# B&R Automation Studio project TD52 (part 71)

#### lIP_EGTCtr.typ
```iecst
TYPE

   tEGTCtr_In : STRUCT
        rT_EG_MaxLim : REAL; (*Exhaust temperature shut down limit from Diane Parameter [°C]*)
        rT_EG_Max : REAL; (*Maximum actual exhaust temperature among all cylinders [°C]*)
        bReset : BOOL; (*Reset of exhaust temperature controller integrator [boolean]*)
        rCA_Init : REAL; (*Reset value of exhaust temperature controller integrator [°CA]*)
        rCA_IP_Act_Rel : REAL; (*External actual ignition timing offset [°CA]*)
    END_STRUCT;

   tEGTCtr_Out : STRUCT
        ulim : REAL; (*Limited controller output [°CA] oldname: ITOffuLim*)
        u : REAL; (*Unlimited controller output [°CA] oldname: ITOffu*)
        up : REAL; (*Unlimited proportional controller output [°CA] oldname: ITOffup*)
        ui : REAL; (*Unlimited integral controller output [°CA] oldname: ITOffui*)
        ud : REAL; (*Unlimited derivative controller output [°CA] oldname: ITOffud*)
        e : REAL; (*Control error without anti-windup [°C] oldname: ITOffe*)
        AW : REAL; (*Anti-windup feedback error [°C] oldname: ITOffAW*)
    END_STRUCT;

   tEGTCtr_Perm : STRUCT
        rT_EG_DltLim : REAL; (*Delta margin from exhaust temperature limit [°C] oldname: TExhLimCntMar*)
        Kp : REAL; (*Proportional gain of exhaust limit controller [°CA/°C]*)
        Ki : REAL; (*Integral gain of exhaust limit controller [°CA/°C/s]*)
        Kd : REAL; (*Derivative gain of exhaust limit controller [°CA*s/°C]*)
        N : REAL; (*Filter constant for derivative controller gain [1/s]*)
        UpLim : REAL; (*Upper limit for controller output [CAD]*)
        LoLim : REAL; (*Lower limit for controller output [°CA]*)
        KAW : REAL; (*Anti windup gain for exhaust temperature controller integrator [°C/°CA]*)
        DeadLoD : REAL; (*Lower deadband limit for derivative part [°C]*)
        DeadUpD : REAL; (*Upper deadband limit for derivative part [°C]*)
    END_STRUCT;
END_TYPE
TYPE
BlockIO_IP_EGTCtr : STRUCT
	perm : tEGTCtr_Perm;
	BusCreator : tEGTCtr_Out;
	in : tEGTCtr_In;
END_STRUCT;
D_Work_IP_EGTCtr : STRUCT
	DiscreteTimeIntegrator_DSTATE : REAL;
	DiscreteTimeIntegrator1_DSTATE : REAL;
	DiscreteTimeIntegrator_PrevRese : SINT;
	DiscreteTimeIntegrator1_PrevRes : SINT;
	DiscreteTimeIntegrator_IC_LOADI : USINT;
END_STRUCT;
END_TYPE
```

#### IP_EGTCtr.h
```c
/********************************************************************
 * COPYRIGHT -- Bernecker + Rainer Industrie-Elektronik Ges.m.b.H.
 ********************************************************************
 * Program: IP_EGTCtr
 * File: IP_EGTCtr.h
 * Author: 302013638
 * Created: Fri Sep 10 20:20:48 2010
 ********************************************************************
 * Header for program IP_EGTCtr
 ********************************************************************
 * Generated with B&R Automation Studio Target for Simulink V4.2
 * (ERT based)
 ********************************************************************/

#ifndef RTW_HEADER_IP_EGTCtr_h_
#define RTW_HEADER_IP_EGTCtr_h_
#ifndef IP_EGTCtr_COMMON_INCLUDES_
# define IP_EGTCtr_COMMON_INCLUDES_
#include "rtwtypes.h"
#endif                                 /* IP_EGTCtr_COMMON_INCLUDES_ */

#include "IP_EGTCtr_types.h"
#include "lIP_EGTCtr.h"

/* Macros for accessing real-time model data structure */
#ifndef rtmGetErrorStatus
# define rtmGetErrorStatus(rtm)        ((void*) 0)
#endif

#ifndef rtmSetErrorStatus
# define rtmSetErrorStatus(rtm, val)   ((void) 0)
#endif

#ifndef rtmGetStopRequested
# define rtmGetStopRequested(rtm)      ((void*) 0)
#endif

#ifndef MIN
#define MIN(a,b)                       ((a) < (b) ? (a) : (b))
#endif

#ifndef MAX
#define MAX(a,b)                       ((a) > (b) ? (a) : (b))
#endif

/* Block signals (auto storage) */

/* Block states (auto storage) for system '<Root>' */

/* Block signals (auto storage) */
extern BlockIO_IP_EGTCtr IP_EGTCtr_B;

/* Block states (auto storage) */
extern D_Work_IP_EGTCtr IP_EGTCtr_DWork;

/* Model entry point functions */
extern void IP_EGTCtr_initialize(struct fIP_EGTCtr* inst);
extern void IP_EGTCtr_step(struct fIP_EGTCtr* inst);
extern void IP_EGTCtr_terminate(struct fIP_EGTCtr* inst);

/*-
 * The generated code includes comments that allow you to trace directly
 * back to the appropriate location in the model.  The basic format
 * is <system>/block_name, where system is the system number (uniquely
 * assigned by Simulink) and block_name is the name of the block.
 *
 * Use the MATLAB hilite_system command to trace the generated code back
 * to the model.  For example,
 *
 * hilite_system('<S3>')    - opens system 3
 * hilite_system('<S3>/Kp') - opens and selects block Kp which resides in S3
 *
 * Here is the system hierarchy for this model
 *
 * '<Root>' : 'IP_EGTCtr'
 * '<S1>'   : 'IP_EGTCtr/DocBlock'
 * '<S2>'   : 'IP_EGTCtr/Model Info'
 * '<S3>'   : 'IP_EGTCtr/TexhCntrSys'
 * '<S4>'   : 'IP_EGTCtr/TexhCntrSys/Dead Zone Dynamic'
 * '<S5>'   : 'IP_EGTCtr/TexhCntrSys/Saturation Dynamic4'
 */
#endif                                 /* RTW_HEADER_IP_EGTCtr_h_ */
```

#### IP_EGTCtr_private.h
```c
/********************************************************************
 * COPYRIGHT -- Bernecker + Rainer Industrie-Elektronik Ges.m.b.H.
 ********************************************************************
 * Program: IP_EGTCtr
 * File: IP_EGTCtr_private.h
 * Author: 302013638
 * Created: Fri Sep 10 20:20:48 2010
 ********************************************************************
 * Header for program IP_EGTCtr
 ********************************************************************
 * Generated with B&R Automation Studio Target for Simulink V4.2
 * (ERT based)
 ********************************************************************/

#ifndef RTW_HEADER_IP_EGTCtr_private_h_
#define RTW_HEADER_IP_EGTCtr_private_h_
#include "rtwtypes.h"
#include <bur/plctypes.h>
#ifndef __RTWTYPES_H__
#error This file requires rtwtypes.h to be included
#else
#ifdef TMWTYPES_PREVIOUSLY_INCLUDED
#error This file requires rtwtypes.h to be included before tmwtypes.h
#else

/* Check for inclusion of an incorrect version of rtwtypes.h */
#ifndef RTWTYPES_ID_C08S16I32L32N32F1
#error This code was generated with a different "rtwtypes.h" than the file included
#endif                                 /* RTWTYPES_ID_C08S16I32L32N32F1 */
#endif                                 /* TMWTYPES_PREVIOUSLY_INCLUDED */
#endif                                 /* __RTWTYPES_H__ */

#ifndef MIN
#define MIN(a,b)                       ((a) < (b) ? (a) : (b))
#endif

#ifndef MAX
#define MAX(a,b)                       ((a) > (b) ? (a) : (b))
#endif
#endif                                 /* RTW_HEADER_IP_EGTCtr_private_h_ */
```

#### IP_EGTCtr_types.h
```c
/********************************************************************
 * COPYRIGHT -- Bernecker + Rainer Industrie-Elektronik Ges.m.b.H.
 ********************************************************************
 * Program: IP_EGTCtr
 * File: IP_EGTCtr_types.h
 * Author: 302013638
 * Created: Fri Sep 10 20:20:48 2010
 ********************************************************************
 * Header for program IP_EGTCtr
 ********************************************************************
 * Generated with B&R Automation Studio Target for Simulink V4.2
 * (ERT based)
 ********************************************************************/

#ifndef RTW_HEADER_IP_EGTCtr_types_h_
#define RTW_HEADER_IP_EGTCtr_types_h_
#include "rtwtypes.h"
#ifndef MIN
#define MIN(a,b)                       ((a) < (b) ? (a) : (b))
#endif

#ifndef MAX
#define MAX(a,b)                       ((a) > (b) ? (a) : (b))
#endif

#endif                                 /* RTW_HEADER_IP_EGTCtr_types_h_ */
```

#### rtwtypes.h
```c
/********************************************************************
 * COPYRIGHT -- Bernecker + Rainer Industrie-Elektronik Ges.m.b.H.
 ********************************************************************
 * Program: IP_EGTCtr
 * File: rtwtypes.h
 * Author: 302013638
 * Created: Fri Sep 10 20:20:48 2010
 ********************************************************************
 * Header for program IP_EGTCtr
 ********************************************************************
 * Generated with B&R Automation Studio Target for Simulink V4.2
 * (ERT based)
 ********************************************************************/

#ifndef __RTWTYPES_H__
#define __RTWTYPES_H__
#ifndef TRUE
# define TRUE                          (1U)
#endif

#ifndef FALSE
# define FALSE                         (0U)
#endif

#ifndef __TMWTYPES__
#define __TMWTYPES__
#include <limits.h>

/*=======================================================================*
 * Target hardware information
 *   Device type: Intel->x86/Pentium
 *   Number of bits:     char:   8    short:   16    long:  32
 *                       long:  32
 *                       native word size:  32
 *   Byte ordering: LittleEndian
 *   Signed integer division rounds to: Zero
 *   Shift right on a signed integer as arithmetic shift: on
 *=======================================================================*/

/*=======================================================================*
 * Fixed width word size data types:                                     *
 *   int8_T, int16_T, int32_T     - signed 8, 16, or 32 bit integers     *
 *   uint8_T, uint16_T, uint32_T  - unsigned 8, 16, or 32 bit integers   *
 *   real32_T, real64_T           - 32 and 64 bit floating point numbers *
 *=======================================================================*/
typedef signed char int8_T;
typedef unsigned char uint8_T;
typedef short int16_T;
typedef unsigned short uint16_T;
typedef long int32_T;
typedef unsigned long uint32_T;
typedef float real32_T;
typedef double real64_T;

/*===========================================================================*
 * Generic type definitions: real_T, time_T, boolean_T, int_T, uint_T,       *
 *                           ulong_T, char_T and byte_T.                     *
 *===========================================================================*/
typedef double real_T;
typedef double time_T;
typedef unsigned char boolean_T;
typedef long int_T;
typedef unsigned long uint_T;
typedef unsigned long ulong_T;
typedef char char_T;
typedef unsigned char uchar_T;
typedef char_T byte_T;

/*=======================================================================*
 * Min and Max:                                                          *
 *   int8_T, int16_T, int32_T     - signed 8, 16, or 32 bit integers     *
 *   uint8_T, uint16_T, uint32_T  - unsigned 8, 16, or 32 bit integers   *
 *=======================================================================*/
#define MAX_int8_T                     ((int8_T)(127))
#define MIN_int8_T                     ((int8_T)(-128))
#define MAX_uint8_T                    ((uint8_T)(255U))
#define MIN_uint8_T                    ((uint8_T)(0U))
#define MAX_int16_T                    ((int16_T)(32767))
#define MIN_int16_T                    ((int16_T)(-32768))
#define MAX_uint16_T                   ((uint16_T)(65535U))
#define MIN_uint16_T                   ((uint16_T)(0U))
#define MAX_int32_T                    ((int32_T)(2147483647))
#define MIN_int32_T                    ((int32_T)(-2147483647-1))
#define MAX_uint32_T                   ((uint32_T)(0xFFFFFFFFU))
#define MIN_uint32_T                   ((uint32_T)(0U))

/* Logical type definitions */
#if (!defined(__cplusplus)) && (!defined(__true_false_are_keywords))
#  ifndef false
#   define false                       (0U)
#  endif

#  ifndef true
#   define true                        (1U)
#  endif
#endif

/*
 * Simulink Coder assumes the code is compiled on a target using a 2's complement representation
 * for signed integer values.
 */
#if ((SCHAR_MIN + 1) != -SCHAR_MAX)
#error "This code must be compiled using a 2's complement representation for signed integer values"
#endif

/* This ID is used to detect inclusion of an incompatible rtwtypes.h */
#define RTWTYPES_ID_C08S16I32L32N32F1
#else                                  /* __TMWTYPES__ */
#define TMWTYPES_PREVIOUSLY_INCLUDED
#endif                                 /* __TMWTYPES__ */

/* Block D-Work pointer type */
typedef void * pointer_T;

/* Simulink specific types */
#ifndef __SIMSTRUC_TYPES_H__
#define __SIMSTRUC_TYPES_H__

/* Trigger directions: falling, either, and rising */
typedef enum {
  FALLING_ZERO_CROSSING = -1,
  ANY_ZERO_CROSSING = 0,
  RISING_ZERO_CROSSING = 1
} ZCDirection;

/* Previous state of a trigger signal */
typedef uint8_T ZCSigState;

/* Initial value of a trigger zero crossing signal */
#define UNINITIALIZED_ZCSIG            0x03U
#define NEG_ZCSIG                      0x02U
#define POS_ZCSIG                      0x01U
#define ZERO_ZCSIG                     0x00U

/* Current state of a trigger signal */
typedef enum {
  FALLING_ZCEVENT = -1,
  NO_ZCEVENT = 0,
  RISING_ZCEVENT = 1
} ZCEventType;

#endif                                 /* __SIMSTRUC_TYPES_H__ */
#endif                                 /* __RTWTYPES_H__ */

#ifndef MIN
#define MIN(a,b)                       ((a) < (b) ? (a) : (b))
#endif

#ifndef MAX
#define MAX(a,b)                       ((a) > (b) ? (a) : (b))
#endif
```

#### IP_EGTCtr.c
```c
/********************************************************************
 * COPYRIGHT -- Bernecker + Rainer Industrie-Elektronik Ges.m.b.H.
 ********************************************************************
 * Program: IP_EGTCtr
 * File: IP_EGTCtr.c
 * Author: 302013638
 * Created: Fri Sep 10 20:20:48 2010
 ********************************************************************
 * Implementation of program IP_EGTCtr
 ********************************************************************
 * Generated with B&R Automation Studio Target for Simulink V4.2
 * (ERT based)
 ********************************************************************/
#include "IP_EGTCtr.h"
#include "IP_EGTCtr_private.h"

/*  Defines */

/*  Data Types */

/**************************** GLOBAL DATA *************************************/
/*  Definitions */

/* Block signals (auto storage) */
struct BlockIO_IP_EGTCtr IP_EGTCtr_B;

/* Block states (auto storage) */
struct D_Work_IP_EGTCtr IP_EGTCtr_DWork;

/*  Declarations  */

/***************************** FILE SCOPE DATA ********************************/

/*************************** FUNCTIONS ****************************************/

/* Model step function */
void IP_EGTCtr_step(struct fIP_EGTCtr* inst)
{
  /* local block i/o variables */
  boolean_T rtb_bReset;
  real32_T rtb_e;
  real32_T rtb_up;
  real32_T rtb_ud;
  real32_T rtb_Product2;
  real32_T rtb_Add;

  /* S-Function (bur_bus_in): '<Root>/Bus Input2' */
  IP_EGTCtr_B.in = inst->in;

  /* BusSelector: '<Root>/BusConversion_InsertedFor_Bus Creator1_at_inport_1' */
  rtb_bReset = IP_EGTCtr_B.in.bReset;

  /* S-Function (bur_bus_in): '<Root>/Bus Input1' */
  IP_EGTCtr_B.perm = inst->perm;

  /* Gain: '<S3>/Gain' incorporates:
   *  Sum: '<S3>/Add4'
   *  Sum: '<S3>/Add6'
   */
  rtb_e = -((IP_EGTCtr_B.in.rT_EG_MaxLim - IP_EGTCtr_B.perm.rT_EG_DltLim) -
            IP_EGTCtr_B.in.rT_EG_Max);

  /* Product: '<S3>/Product1' */
  rtb_up = rtb_e * IP_EGTCtr_B.perm.Kp;

  /* DiscreteIntegrator: '<S3>/Discrete-Time Integrator' */
  if (IP_EGTCtr_DWork.DiscreteTimeIntegrator_IC_LOADI != 0) {
    IP_EGTCtr_DWork.DiscreteTimeIntegrator_DSTATE = IP_EGTCtr_B.in.rCA_Init;
  }

  if (rtb_bReset || (IP_EGTCtr_DWork.DiscreteTimeIntegrator_PrevRese != 0)) {
    IP_EGTCtr_DWork.DiscreteTimeIntegrator_DSTATE = IP_EGTCtr_B.in.rCA_Init;
  }

  /* DiscreteIntegrator: '<S3>/Discrete-Time Integrator1' */
  if (rtb_bReset || (IP_EGTCtr_DWork.DiscreteTimeIntegrator1_PrevRes != 0)) {
    IP_EGTCtr_DWork.DiscreteTimeIntegrator1_DSTATE = 0.0F;
  }

  /* Switch: '<S4>/Switch' incorporates:
   *  RelationalOperator: '<S4>/u_GTE_up'
   *  RelationalOperator: '<S4>/u_GT_lo'
   *  Switch: '<S4>/Switch1'
   */
  if (rtb_e >= IP_EGTCtr_B.perm.DeadUpD) {
    rtb_ud = IP_EGTCtr_B.perm.DeadUpD;
  } else if (rtb_e > IP_EGTCtr_B.perm.DeadLoD) {
    /* Switch: '<S4>/Switch1' */
    rtb_ud = rtb_e;
  } else {
    rtb_ud = IP_EGTCtr_B.perm.DeadLoD;
  }

  /* End of Switch: '<S4>/Switch' */

  /* Product: '<S3>/Divide3' incorporates:
   *  DiscreteIntegrator: '<S3>/Discrete-Time Integrator1'
   *  Product: '<S3>/Product3'
   *  Sum: '<S3>/Sum1'
   *  Sum: '<S4>/Diff'
   */
  rtb_ud = ((rtb_e - rtb_ud) * IP_EGTCtr_B.perm.Kd -
            IP_EGTCtr_DWork.DiscreteTimeIntegrator1_DSTATE) * IP_EGTCtr_B.perm.N;

  /* Sum: '<S3>/Add' incorporates:
   *  DiscreteIntegrator: '<S3>/Discrete-Time Integrator'
   */
  rtb_Add = (rtb_up + IP_EGTCtr_DWork.DiscreteTimeIntegrator_DSTATE) + rtb_ud;

  /* Product: '<S3>/Product2' incorporates:
   *  Sum: '<S3>/Add2'
   */
  rtb_Product2 = (rtb_Add - IP_EGTCtr_B.in.rCA_IP_Act_Rel) *
    IP_EGTCtr_B.perm.KAW;

  /* Switch: '<S3>/Switch' incorporates:
   *  RelationalOperator: '<S5>/LowerRelop1'
   *  RelationalOperator: '<S5>/UpperRelop'
   *  Switch: '<S5>/Switch'
   *  Switch: '<S5>/Switch2'
   */
  if (rtb_bReset) {
    /* BusCreator: '<Root>/Bus Creator' incorporates:
     *  Constant: '<S3>/Constant'
     */
    IP_EGTCtr_B.BusCreator.ulim = 0.0F;
  } else if (rtb_Add > IP_EGTCtr_B.perm.UpLim) {
    /* Switch: '<S5>/Switch2' incorporates:
     *  BusCreator: '<Root>/Bus Creator'
     */
    IP_EGTCtr_B.BusCreator.ulim = IP_EGTCtr_B.perm.UpLim;
  } else if (rtb_Add < IP_EGTCtr_B.perm.LoLim) {
    /* Switch: '<S5>/Switch' incorporates:
     *  BusCreator: '<Root>/Bus Creator'
     *  Switch: '<S5>/Switch2'
     */
    IP_EGTCtr_B.BusCreator.ulim = IP_EGTCtr_B.perm.LoLim;
  } else {
    /* BusCreator: '<Root>/Bus Creator' incorporates:
     *  Switch: '<S5>/Switch'
     *  Switch: '<S5>/Switch2'
     */
    IP_EGTCtr_B.BusCreator.ulim = rtb_Add;
  }

  /* End of Switch: '<S3>/Switch' */

  /* BusCreator: '<Root>/Bus Creator' incorporates:
   *  DiscreteIntegrator: '<S3>/Discrete-Time Integrator'
   */
  IP_EGTCtr_B.BusCreator.u = rtb_Add;
  IP_EGTCtr_B.BusCreator.up = rtb_up;
  IP_EGTCtr_B.BusCreator.ui = IP_EGTCtr_DWork.DiscreteTimeIntegrator_DSTATE;
  IP_EGTCtr_B.BusCreator.ud = rtb_ud;
  IP_EGTCtr_B.BusCreator.e = rtb_e;
  IP_EGTCtr_B.BusCreator.AW = rtb_Product2;

  /* S-Function (bur_bus_out): '<Root>/Bus Output' */
  inst->out = IP_EGTCtr_B.BusCreator;

  /* Product: '<S3>/Product' */
  rtb_e *= IP_EGTCtr_B.perm.Ki;

  /* Update for DiscreteIntegrator: '<S3>/Discrete-Time Integrator' incorporates:
   *  Sum: '<S3>/Add5'
   */
  IP_EGTCtr_DWork.DiscreteTimeIntegrator_IC_LOADI = 0U;
  if (!rtb_bReset) {
    IP_EGTCtr_DWork.DiscreteTimeIntegrator_DSTATE += (rtb_e - rtb_Product2) *
      0.01F;
  }

  if (rtb_bReset) {
    IP_EGTCtr_DWork.DiscreteTimeIntegrator_PrevRese = 1;
  } else {
    IP_EGTCtr_DWork.DiscreteTimeIntegrator_PrevRese = 0;
  }

  /* End of Update for DiscreteIntegrator: '<S3>/Discrete-Time Integrator' */

  /* Update for DiscreteIntegrator: '<S3>/Discrete-Time Integrator1' */
  if (!rtb_bReset) {
    IP_EGTCtr_DWork.DiscreteTimeIntegrator1_DSTATE += 0.01F * rtb_ud;
  }

  if (rtb_bReset) {
    IP_EGTCtr_DWork.DiscreteTimeIntegrator1_PrevRes = 1;
  } else {
    IP_EGTCtr_DWork.DiscreteTimeIntegrator1_PrevRes = 0;
  }

  /* End of Update for DiscreteIntegrator: '<S3>/Discrete-Time Integrator1' */
}

/* Model initialize function */
void IP_EGTCtr_initialize(struct fIP_EGTCtr* inst)
{
  /* InitializeConditions for DiscreteIntegrator: '<S3>/Discrete-Time Integrator' */
  IP_EGTCtr_DWork.DiscreteTimeIntegrator_IC_LOADI = 1U;
}

/* Model terminate function */
void IP_EGTCtr_terminate(struct fIP_EGTCtr* inst)
{
  /* (no terminate code required) */
}

/*======================== TOOL VERSION INFORMATION ==========================*
 * MATLAB 8.0 (R2012b)20-Jul-2012                                             *
 * Simulink 8.0 (R2012b)20-Jul-2012                                           *
 * Simulink Coder 8.3 (R2012b)20-Jul-2012                                     *
 * Embedded Coder 6.3 (R2012b)20-Jul-2012                                     *
 * Stateflow 8.0 (R2012b)20-Jul-2012                                          *
 *============================================================================*/

/*======================= LICENSE IN USE INFORMATION =========================*
 * matlab                                                                     *
 * matlab_coder                                                               *
 * real-time_workshop                                                         *
 * rtw_embedded_coder                                                         *
 * simulink                                                                   *
 *============================================================================*/
```

#### main.c
```c
/********************************************************************
 * COPYRIGHT -- Bernecker + Rainer Industrie-Elektronik Ges.m.b.H.
 ********************************************************************
 * Program: IP_EGTCtr
 * File: main.c
 * Author: 302013638
 * Created: Fri Sep 10 20:20:48 2010
 ********************************************************************
 * Implementation of program IP_EGTCtr
 ********************************************************************
 * Generated with B&R Automation Studio Target for Simulink V4.2
 * (ERT based)
 ********************************************************************/
#include <bur/plctypes.h>
#include "IP_EGTCtr.h"
#include "rtwtypes.h"

/* Defines */
#define SS_TERMINATE 4
#define SS_OUTPUT 3
#define SS_INITIALIZE 2

/*  Data Types */

/**************************** GLOBAL DATA *************************************/
/*  Definitions */

/*  Declarations  */

/***************************** FILE SCOPE DATA ********************************/

/*************************** FUNCTIONS ****************************************/
#ifdef __cplusplus

unsigned long bur_heap_size = 6553500;

#endif

void fIP_EGTCtr(struct fIP_EGTCtr* inst)
{

  switch (inst->ssMethodType)
  {
   case SS_INITIALIZE:
    /* call model initialize function */
    IP_EGTCtr_initialize(inst);
    break;

   case SS_OUTPUT:
    /* call model step function */
    IP_EGTCtr_step(inst);

    break;

   case SS_TERMINATE:
    /* call model terminate function */
    IP_EGTCtr_terminate(inst);
    break;
  }
}

/*****************************************************************************
   Function block sample time: 0.01s
 *****************************************************************************/

/*****************************************************************************
   B&R Automation Studio Target for Simulink Version: A4.4.1 (09-Dec-2014)
 *****************************************************************************/

/*======================== TOOL VERSION INFORMATION ==========================*
 * MATLAB 8.0 (R2012b)20-Jul-2012                                             *
 * Simulink 8.0 (R2012b)20-Jul-2012                                           *
 * Simulink Coder 8.3 (R2012b)20-Jul-2012                                     *
 * Embedded Coder 6.3 (R2012b)20-Jul-2012                                     *
 * Stateflow 8.0 (R2012b)20-Jul-2012                                          *
 *============================================================================*/

/*======================= LICENSE IN USE INFORMATION =========================*
 * matlab                                                                     *
 * matlab_coder                                                               *
 * real-time_workshop                                                         *
 * rtw_embedded_coder                                                         *
 * simulink                                                                   *
 *============================================================================*/
```

#### lib_properties.txt
```
For manual assignment to hardware configuration please
add the following additional include directories:

\Logical\MATLAB_includes\R2012b\

And the following additional build options:

-lm -D MODEL=IP_EGTCtr -D NUMST=1 -D NCSTATES=0 -D HAVESTDIO -D ONESTEPFCN=1 -D TERMFCN=1 -D MAT_FILE=0 -D MULTI_INSTANCE_CODE=0 -D INTEGER_CODE=0 -D MT=0 -D CLASSIC_INTERFACE=0 -D TID01EQ=0
```

### Library Logical/EngineController/Lib_EC/lFSync (ANSIC)

#### lFSync.fun
```iecst
FUNCTION_BLOCK fFSync
  VAR_INPUT
    ssMethodType: SINT;
  END_VAR  VAR_INPUT
        In : tFsync_Inputs; (*Inputs to Fast synch*)
  END_VAR
  VAR_INPUT
        Perm : tFsync_Perm; (**)
  END_VAR
  VAR_INPUT
        Para : tFsync_Para; (*Inputs to Fast synch*)
  END_VAR
 VAR_OUTPUT
        dbg : tFsync_Debug; (**)
  END_VAR
  VAR_OUTPUT
        iSkipCyl : USINT; (**)
  END_VAR
  VAR_OUTPUT
        bEnabled : BOOL := FALSE; (*True..AutoCode running, FALSE..switch to standard controller*)
  END_VAR
  VAR_OUTPUT
        Version : UDINT; (**)
  END_VAR
	VAR
		bur_BlockIO_FSync : BlockIO_FSync;
	END_VAR
	VAR
		bur_D_Work_FSync : D_Work_FSync;
	END_VAR
	VAR
		bur_ExternalOutputs_FSync : ExternalOutputs_FSync;
	END_VAR
END_FUNCTION_BLOCK
```

#### lFSync.typ
```iecst
TYPE

   tFsync_Debug : STRUCT
        iSkipCounter : UINT; (**)
        rSwitchSurf : REAL; (**)
        Sf1 : BOOL; (**)
        Sf2 : BOOL; (**)
        H3 : BOOL; (**)
        H4 : BOOL; (**)
        rSmodSlid : REAL; (**)
        iCounterSwitch : UINT; (**)
        bEna : BOOL; (**)
        iNskip_init : USINT; (**)
        iCtrSel : SINT; (**)
        iNumSkipCyl_P : SINT; (*P-part*)
        rN_Set : REAL; (*Speed set poinnt*)
        rN_Eng : REAL; (*Actual speed*)
    END_STRUCT;

   tFsync_Inputs : STRUCT
        bGCB_ON : BOOL; (*Generator circuit breaker closed*)
        rN_Eng : REAL; (*Engine speed in rpm*)
        rF_MMD : REAL; (*Generator frequency [Hz]*)
        rAng_MMD_Diff : REAL; (*Electric angle in deg.*)
        rF_MMD_BusBar : REAL; (*Bus bar frequency in Hz*)
        rT_EO : REAL; (**)
        iIdx_SyOMSS : INT; (*synchronization operating mode selection
0..OFF
1..MAN
2..AUTO*)
        bReset : BOOL; (*reset library*)
    END_STRUCT;

   tFsync_Para : STRUCT
        rN_Offs_Sync : REAL; (**)
        rF_Nom : REAL; (**)
        rN_EngNom : REAL; (**)
        bFastSync : BOOL; (**)
    END_STRUCT;

   tFsync_Perm : STRUCT
        bSpeedSet_ena : BOOL; (*Select the setpoint (1: constant speed, 0: grid frequency)*)
        iCtrSel : SINT; (*Control selection. 1-Std skip firing. 2-Time optimal 3-Time optimal with constraints. 4-Fuel and time optimal. 5-Modified skip f*)
        rN_SetTol : REAL; (*Speed band for speed regulation (rpm, valid only for standard approach)*)
        iSkipCounterLimit : UINT; (*Dwell time for skip firing (in number of 10ms, valid only for the standard approach)*)
        rAngleSetDeg : REAL; (*Electric angle setpoint (in deg, tuning parameter)*)
        rRelaxAngleDeg : REAL; (*Relaxation band for the electric angle setpoint (in deg, tuning parameter)*)
        rWeightFuel : REAL; (*Weighting (high->time, low->fuel)*)
        rHystOptimal : REAL; (*Band around switching surface (nonnegative >=0)*)
        iNum_SkipMax : USINT; (*Maximum cylinders skipped (<=20)*)
        iNum_SkipMin : USINT; (*Minimum number of cylinders (>=0)*)
        rTi_FiltF : REAL; (*Filter constant for grid frequency [s]*)
        rN_enableNorm : REAL; (*Engine speed normalized to enable fast sync controller [-]*)
        rN_idleNorm : REAL; (*Engine speed normalized to enable fast sync controller [-]*)
        rTi_FastSync : REAL; (*switch over to standard controller after this time [s]*)
        bF_act_ena : BOOL; (*use generator frequency as actual value*)
        rT_Cold : REAL; (**)
        rT_Warm : REAL; (**)
        iNum_SkipCyl_Cold : USINT; (*Init skipped cyl at T_Cold*)
        iNum_SkipCyl_Warm : USINT; (*Init skipped cyl at T_Warm*)
        rGain_P : REAL; (*Gain for P-part [NumSkippedCyl/rpm]*)
        iNum_SkipCylLim_P : SINT; (*Limit for P-part [NumSkippedCyl]*)
        bStdCtrl : BOOL; (*Standard controller enabled in AutoCode*)
    END_STRUCT;
END_TYPE
TYPE
BlockIO_FSync : STRUCT
	BusInput1 : tFsync_Perm;
	BusInput : tFsync_Inputs;
	BusInput2 : tFsync_Para;
	UnitDelay : UDINT;
	bEnabled : BOOL;
END_STRUCT;
D_Work_FSync : STRUCT
	DiscreteTimeIntegrator_DSTATE : REAL;
	UnitDelay_DSTATE : UDINT;
	rN_Set_old : REAL;
	skipcounter : UINT;
	Count_Switch : UINT;
	DiscreteTimeIntegrator_PrevRese : SINT;
	DiscreteTimeIntegrator_IC_LOADI : USINT;
	cyl_skipped : USINT;
	ssr : BOOL;
	ssr_Set : BOOL;
	cyl_skipped_not_empty : BOOL;
	bSkipDrehz_O : BOOL;
	bSkipDrehz_U : BOOL;
	No_Access : BOOL;
END_STRUCT;
ExternalInputs_FSync : STRUCT
	In : tFsync_Inputs;
	Para : tFsync_Para;
	Perm : tFsync_Perm;
END_STRUCT;
ExternalOutputs_FSync : STRUCT
	SkipCyl : USINT;
	dbg : tFsync_Debug;
END_STRUCT;
END_TYPE
```

#### FSync.h
```c
/********************************************************************
 * COPYRIGHT -- Bernecker + Rainer Industrie-Elektronik Ges.m.b.H.
 ********************************************************************
 * Program: FSync
 * File: FSync.h
 * Author: 105051359
 * Created: Mon Mar 13 15:42:43 2017
 ********************************************************************
 * Header for program FSync
 ********************************************************************
 * Generated with B&R Automation Studio Target for Simulink V4.2
 * (ERT based)
 ********************************************************************/

#ifndef RTW_HEADER_FSync_h_
#define RTW_HEADER_FSync_h_
#ifndef FSync_COMMON_INCLUDES_
# define FSync_COMMON_INCLUDES_
#include <math.h>
#include "rtwtypes.h"
#endif                                 /* FSync_COMMON_INCLUDES_ */

#include "FSync_types.h"
#include "lFSync.h"

/* Macros for accessing real-time model data structure */
#ifndef rtmGetErrorStatus
# define rtmGetErrorStatus(rtm)        ((void*) 0)
#endif

#ifndef rtmSetErrorStatus
# define rtmSetErrorStatus(rtm, val)   ((void) 0)
#endif

#ifndef rtmGetStopRequested
# define rtmGetStopRequested(rtm)      ((void*) 0)
#endif

#ifndef MIN
#define MIN(a,b)                       ((a) < (b) ? (a) : (b))
#endif

#ifndef MAX
#define MAX(a,b)                       ((a) > (b) ? (a) : (b))
#endif

/* user code (top of header file) */
/***************************************************************************************************
 * COPYRIGHT -- INNIO Jenbacher GmbH & CO OG
 ****************************************************************************************************
 * Program:            FSync
 * Author:             arnolge00
 * Created:            05.07.2021 14:02
 ****************************************************************************************************
 * MODEL INFORMATION
 ****************************************************************************************************
 * Model Name:         C:\Users\arnolge00\Documents\MATLAB\Git\FastSync\03_Simulation\ModelFull\FSync.slx
 * Model Version:      0.07
 * Simulink Version:   R2012b
 * B&R Target:         V4.5.1
 * Description:
 ****************************************************************************************************
 * HISTORY
 ****************************************************************************************************
 * Last Modified By:   arnolge00
 * Last Modified Date: Mon Jul 05 14:00:19 2021
 * Modified Comment:   V0.01    11.05.2017    Arnold,   first version used @P20
 *                     V0.02    23.05.2017    Arnold,   Generator frequency included
 *                     V0.03    29.05.2017    Arnold,   added idle speed
 *                     V0.04    29.05.2017    Arnold,   added P-part and Sync offset for Ctrl=1
 *                     V0.05    05.08.2020    Schmidt,  changed grid frequency variable from rF_MMD_Synch2 to rF_MMD_BusBar
 *                     V0.06    25.01.2021    Schmidt,  use of frequency based speed set-point (rN_Set) only if rF_MMD_BusBar > 0.5*rF_Nom
 *                     V0.07    05.07.2021    Arnold,   prevent NaN with using of standard filter
 ****************************************************************************************************/

/* Block signals (auto storage) */

/* Block states (auto storage) for system '<Root>' */

/* External inputs (root inport signals with auto storage) */

/* External outputs (root outports fed by signals with auto storage) */

/* Model entry point functions */
extern void FSync_initialize(D_Work_FSync *FSync_DWork, struct fFSync* inst);
extern void FSync_step(BlockIO_FSync *FSync_B, D_Work_FSync *FSync_DWork,
  ExternalOutputs_FSync *FSync_Y, struct fFSync* inst);
extern void FSync_terminate(struct fFSync* inst);

/*-
 * The generated code includes comments that allow you to trace directly
 * back to the appropriate location in the model.  The basic format
 * is <system>/block_name, where system is the system number (uniquely
 * assigned by Simulink) and block_name is the name of the block.
 *
 * Use the MATLAB hilite_system command to trace the generated code back
 * to the model.  For example,
 *
 * hilite_system('<S3>')    - opens system 3
 * hilite_system('<S3>/Kp') - opens and selects block Kp which resides in S3
 *
 * Here is the system hierarchy for this model
 *
 * '<Root>' : 'FSync'
 * '<S1>'   : 'FSync/Environment Controller'
 * '<S2>'   : 'FSync/Environment Controller1'
 * '<S3>'   : 'FSync/Environment Controller2'
 * '<S4>'   : 'FSync/Info'
 * '<S5>'   : 'FSync/NSkipInit'
 * '<S6>'   : 'FSync/SkipFireCtrl'
 * '<S7>'   : 'FSync/Skipfire_active'
 * '<S8>'   : 'FSync/Time2Sample'
 * '<S9>'   : 'FSync/ValueSelect'
 * '<S10>'  : 'FSync/ValueSelect/Compare To Constant1'
 * '<S11>'  : 'FSync/ValueSelect/Compare To Zero1'
 * '<S12>'  : 'FSync/ValueSelect/Compare To Zero2'
 * '<S13>'  : 'FSync/ValueSelect/Compare To Zero3'
 * '<S14>'  : 'FSync/ValueSelect/Compare To Zero4'
 * '<S15>'  : 'FSync/ValueSelect/Divisor'
 * '<S16>'  : 'FSync/ValueSelect/Divisor1'
 * '<S17>'  : 'FSync/ValueSelect/Filter'
 * '<S18>'  : 'FSync/ValueSelect/Saturation Dynamic'
 * '<S19>'  : 'FSync/ValueSelect/Divisor/Data Type Conversion Inherited'
 * '<S20>'  : 'FSync/ValueSelect/Divisor1/Data Type Conversion Inherited'
 * '<S21>'  : 'FSync/ValueSelect/Filter/Divisor'
 * '<S22>'  : 'FSync/ValueSelect/Filter/Divisor/Data Type Conversion Inherited'
 */
#endif                                 /* RTW_HEADER_FSync_h_ */
```

#### FSync_private.h
```c
/********************************************************************
 * COPYRIGHT -- Bernecker + Rainer Industrie-Elektronik Ges.m.b.H.
 ********************************************************************
 * Program: FSync
 * File: FSync_private.h
 * Author: 105051359
 * Created: Mon Mar 13 15:42:43 2017
 ********************************************************************
 * Header for program FSync
 ********************************************************************
 * Generated with B&R Automation Studio Target for Simulink V4.2
 * (ERT based)
 ********************************************************************/

#ifndef RTW_HEADER_FSync_private_h_
#define RTW_HEADER_FSync_private_h_
#include "rtwtypes.h"
#include <bur/plctypes.h>
#ifndef UCHAR_MAX
#include <limits.h>
#endif

#if ( UCHAR_MAX != (0xFFU) ) || ( SCHAR_MAX != (0x7F) )
#error "Code was generated for compiler with different sized uchar/char. Consider adjusting Emulation Hardware word size settings on the Hardware Implementation pane to match your compiler word sizes as defined in the compiler's limits.h header file. Alternatively, you can select 'None' for Emulation Hardware and select the 'Enable portable word sizes' option for ERT based targets, which will disable the preprocessor word size checks."
#endif

#if ( USHRT_MAX != (0xFFFFU) ) || ( SHRT_MAX != (0x7FFF) )
#error "Code was generated for compiler with different sized ushort/short. Consider adjusting Emulation Hardware word size settings on the Hardware Implementation pane to match your compiler word sizes as defined in the compilers limits.h header file. Alternatively, you can select 'None' for Emulation Hardware and select the 'Enable portable word sizes' option for ERT based targets, this will disable the preprocessor word size checks."
#endif

#if ( UINT_MAX != (0xFFFFFFFFU) ) || ( INT_MAX != (0x7FFFFFFF) )
#error "Code was generated for compiler with different sized uint/int. Consider adjusting Emulation Hardware word size settings on the Hardware Implementation pane to match your compiler word sizes as defined in the compilers limits.h header file. Alternatively, you can select 'None' for Emulation Hardware and select the 'Enable portable word sizes' option for ERT based targets, this will disable the preprocessor word size checks."
#endif

#if ( ULONG_MAX != (0xFFFFFFFFU) ) || ( LONG_MAX != (0x7FFFFFFF) )
#error "Code was generated for compiler with different sized ulong/long. Consider adjusting Emulation Hardware word size settings on the Hardware Implementation pane to match your compiler word sizes as defined in the compilers limits.h header file. Alternatively, you can select 'None' for Emulation Hardware and select the 'Enable portable word sizes' option for ERT based targets, this will disable the preprocessor word size checks."
#endif

#ifndef __RTWTYPES_H__
#error This file requires rtwtypes.h to be included
#else
#ifdef TMWTYPES_PREVIOUSLY_INCLUDED
#error This file requires rtwtypes.h to be included before tmwtypes.h
#else

/* Check for inclusion of an incorrect version of rtwtypes.h */
#ifndef RTWTYPES_ID_C08S16I32L32N32F1
#error This code was generated with a different "rtwtypes.h" than the file included
#endif                                 /* RTWTYPES_ID_C08S16I32L32N32F1 */
#endif                                 /* TMWTYPES_PREVIOUSLY_INCLUDED */
#endif                                 /* __RTWTYPES_H__ */

#ifndef MIN
#define MIN(a,b)                       ((a) < (b) ? (a) : (b))
#endif

#ifndef MAX
#define MAX(a,b)                       ((a) > (b) ? (a) : (b))
#endif

void BINARYSEARCH_S16(uint32_T *piLeft, uint32_T *piRght, int16_T u, const
                      int16_T *pData, uint32_T iHi, struct fFSync* inst);
void INTERPOLATE_U8S16_S16(uint8_T *pY, int16_T yL, int16_T yR, int16_T x,
  int16_T xL, int16_T xR, struct fFSync* inst);
void LookUp_U8S16_S16(uint8_T *pY, const int16_T *pYData, int16_T u, const
                      int16_T *pUData, uint32_T iHi, struct fFSync* inst);
extern int32_T div_s32_floor(int32_T numerator, int32_T denominator, struct fFSync* inst);

#endif                                 /* RTW_HEADER_FSync_private_h_ */
```

#### FSync_types.h
```c
/********************************************************************
 * COPYRIGHT -- Bernecker + Rainer Industrie-Elektronik Ges.m.b.H.
 ********************************************************************
 * Program: FSync
 * File: FSync_types.h
 * Author: 105051359
 * Created: Mon Mar 13 15:42:43 2017
 ********************************************************************
 * Header for program FSync
 ********************************************************************
 * Generated with B&R Automation Studio Target for Simulink V4.2
 * (ERT based)
 ********************************************************************/

#ifndef RTW_HEADER_FSync_types_h_
#define RTW_HEADER_FSync_types_h_
#include "rtwtypes.h"
#ifndef MIN
#define MIN(a,b)                       ((a) < (b) ? (a) : (b))
#endif

#ifndef MAX
#define MAX(a,b)                       ((a) > (b) ? (a) : (b))
#endif

#endif                                 /* RTW_HEADER_FSync_types_h_ */
```

#### rtwtypes.h
```c
/********************************************************************
 * COPYRIGHT -- Bernecker + Rainer Industrie-Elektronik Ges.m.b.H.
 ********************************************************************
 * Program: FSync
 * File: rtwtypes.h
 * Author: 105051359
 * Created: Mon Mar 13 15:42:43 2017
 ********************************************************************
 * Header for program FSync
 ********************************************************************
 * Generated with B&R Automation Studio Target for Simulink V4.2
 * (ERT based)
 ********************************************************************/

#ifndef __RTWTYPES_H__
#define __RTWTYPES_H__
#ifndef TRUE
# define TRUE                          (1U)
#endif

#ifndef FALSE
# define FALSE                         (0U)
#endif

#ifndef __TMWTYPES__
#define __TMWTYPES__
#include <limits.h>

/*=======================================================================*
 * Target hardware information
 *   Device type: Intel->x86/Pentium
 *   Number of bits:     char:   8    short:   16    long:  32
 *                       long:  32
 *                       native word size:  32
 *   Byte ordering: LittleEndian
 *   Signed integer division rounds to: Zero
 *   Shift right on a signed integer as arithmetic shift: on
 *=======================================================================*/

/*=======================================================================*
 * Fixed width word size data types:                                     *
 *   int8_T, int16_T, int32_T     - signed 8, 16, or 32 bit integers     *
 *   uint8_T, uint16_T, uint32_T  - unsigned 8, 16, or 32 bit integers   *
 *   real32_T, real64_T           - 32 and 64 bit floating point numbers *
 *=======================================================================*/
typedef signed char int8_T;
typedef unsigned char uint8_T;
typedef short int16_T;
typedef unsigned short uint16_T;
typedef long int32_T;
typedef unsigned long uint32_T;
typedef float real32_T;
typedef double real64_T;

/*===========================================================================*
 * Generic type definitions: real_T, time_T, boolean_T, int_T, uint_T,       *
 *                           ulong_T, char_T and byte_T.                     *
 *===========================================================================*/
typedef double real_T;
typedef double time_T;
typedef unsigned char boolean_T;
typedef long int_T;
typedef unsigned long uint_T;
typedef unsigned long ulong_T;
typedef char char_T;
typedef unsigned char uchar_T;
typedef char_T byte_T;

/*=======================================================================*
 * Min and Max:                                                          *
 *   int8_T, int16_T, int32_T     - signed 8, 16, or 32 bit integers     *
 *   uint8_T, uint16_T, uint32_T  - unsigned 8, 16, or 32 bit integers   *
 *=======================================================================*/
#define MAX_int8_T                     ((int8_T)(127))
#define MIN_int8_T                     ((int8_T)(-128))
#define MAX_uint8_T                    ((uint8_T)(255U))
#define MIN_uint8_T                    ((uint8_T)(0U))
#define MAX_int16_T                    ((int16_T)(32767))
#define MIN_int16_T                    ((int16_T)(-32768))
#define MAX_uint16_T                   ((uint16_T)(65535U))
#define MIN_uint16_T                   ((uint16_T)(0U))
#define MAX_int32_T                    ((int32_T)(2147483647))
#define MIN_int32_T                    ((int32_T)(-2147483647-1))
#define MAX_uint32_T                   ((uint32_T)(0xFFFFFFFFU))
#define MIN_uint32_T                   ((uint32_T)(0U))

/* Logical type definitions */
#if (!defined(__cplusplus)) && (!defined(__true_false_are_keywords))
#  ifndef false
#   define false                       (0U)
#  endif

#  ifndef true
#   define true                        (1U)
#  endif
#endif

/*
 * Simulink Coder assumes the code is compiled on a target using a 2's complement representation
 * for signed integer values.
 */
#if ((SCHAR_MIN + 1) != -SCHAR_MAX)
#error "This code must be compiled using a 2's complement representation for signed integer values"
#endif

/* This ID is used to detect inclusion of an incompatible rtwtypes.h */
#define RTWTYPES_ID_C08S16I32L32N32F1
#else                                  /* __TMWTYPES__ */
#define TMWTYPES_PREVIOUSLY_INCLUDED
#endif                                 /* __TMWTYPES__ */

/* Block D-Work pointer type */
typedef void * pointer_T;

/* Simulink specific types */
#ifndef __SIMSTRUC_TYPES_H__
#define __SIMSTRUC_TYPES_H__

/* Trigger directions: falling, either, and rising */
typedef enum {
  FALLING_ZERO_CROSSING = -1,
  ANY_ZERO_CROSSING = 0,
  RISING_ZERO_CROSSING = 1
} ZCDirection;

/* Previous state of a trigger signal */
typedef uint8_T ZCSigState;

/* Initial value of a trigger zero crossing signal */
#define UNINITIALIZED_ZCSIG            0x03U
#define NEG_ZCSIG                      0x02U
#define POS_ZCSIG                      0x01U
#define ZERO_ZCSIG                     0x00U

/* Current state of a trigger signal */
typedef enum {
  FALLING_ZCEVENT = -1,
  NO_ZCEVENT = 0,
  RISING_ZCEVENT = 1
} ZCEventType;

#endif                                 /* __SIMSTRUC_TYPES_H__ */
#endif                                 /* __RTWTYPES_H__ */

#ifndef MIN
#define MIN(a,b)                       ((a) < (b) ? (a) : (b))
#endif

#ifndef MAX
#define MAX(a,b)                       ((a) > (b) ? (a) : (b))
#endif
```

#### FSync.c
```c
/********************************************************************
 * COPYRIGHT -- Bernecker + Rainer Industrie-Elektronik Ges.m.b.H.
 ********************************************************************
 * Program: FSync
 * File: FSync.c
 * Author: 105051359
 * Created: Mon Mar 13 15:42:43 2017
 ********************************************************************
 * Implementation of program FSync
 ********************************************************************
 * Generated with B&R Automation Studio Target for Simulink V4.2
 * (ERT based)
 ********************************************************************/
#include "FSync.h"
#include "FSync_private.h"

/*  Defines */

/*  Data Types */

/**************************** GLOBAL DATA *************************************/
/*  Definitions */

/*  Declarations  */

/***************************** FILE SCOPE DATA ********************************/

/*************************** FUNCTIONS ****************************************/

/* Lookup Binary Search Utility BINARYSEARCH_S16 */
void BINARYSEARCH_S16(uint32_T *piLeft, uint32_T *piRght, int16_T u, const
                      int16_T *pData, uint32_T iHi, struct fFSync* inst)
{
  /* Find the location of current input value in the data table. */
  *piLeft = 0U;
  *piRght = iHi;
  if (u <= pData[0] ) {
    /* Less than or equal to the smallest point in the table. */
    *piRght = 0U;
  } else if (u >= pData[iHi] ) {
    /* Greater than or equal to the largest point in the table. */
    *piLeft = iHi;
  } else {
    uint32_T i;

    /* Do a binary search. */
    while (( *piRght - *piLeft ) > 1U ) {
      /* Get the average of the left and right indices using to Floor rounding. */
      i = (*piLeft + *piRght) >> 1;

      /* Move either the right index or the left index so that */
      /*  LeftDataPoint <= CurrentValue < RightDataPoint */
      if (u < pData[i] ) {
        *piRght = i;
      } else {
        *piLeft = i;
      }
    }
  }
}

/* Lookup Interpolation INTERPOLATE_U8S16_S16 */
void INTERPOLATE_U8S16_S16(uint8_T *pY, int16_T yL, int16_T yR, int16_T x,
  int16_T xL, int16_T xR, struct fFSync* inst)
{
  int32_T bigProd;
  int16_T yDiff;
  int16_T xNum;
  int16_T xDen;
  uint8_T yAdjust;
  *pY = (uint8_T)yL;

  /* If x is not strictly between xR and xL
   * then an interpolation calculation is not necessary x == xL
   * or not valid.  The invalid situation is expected when the input
   * is beyond the left or right end of the table.  The design is
   * that yL holds the correct value for *pY
   * in invalid situations.
   */
  if ((xR > xL) && (x > xL) ) {
    xDen = xR;
    xDen = (int16_T)(xDen - xL);
    xNum = x;
    xNum = (int16_T)(xNum - xL);
    if (yR >= yL ) {
      yDiff = yR;
      yDiff = (int16_T)(yDiff - yL);
    } else {
      yDiff = yL;
      yDiff = (int16_T)(yDiff - yR);
    }

    bigProd = yDiff * xNum;
    yAdjust = (uint8_T)div_s32_floor(bigProd, (int32_T)xDen, inst);
    if (yR >= yL ) {
      *pY = (uint8_T)((uint32_T)*pY + (uint32_T)yAdjust);
    } else {
      *pY = (uint8_T)((uint32_T)*pY - (uint32_T)yAdjust);
    }
  }
}

/* Lookup Utility LookUp_U8S16_S16 */
void LookUp_U8S16_S16(uint8_T *pY, const int16_T *pYData, int16_T u, const
                      int16_T *pUData, uint32_T iHi, struct fFSync* inst)
{
  uint32_T iLeft;
  uint32_T iRght;
  BINARYSEARCH_S16( &(iLeft), &(iRght), u, pUData, iHi, inst);
  INTERPOLATE_U8S16_S16( pY, pYData[iLeft], pYData[iRght], u, pUData[iLeft],
                        pUData[iRght], inst);
}

int32_T div_s32_floor(int32_T numerator, int32_T denominator, struct fFSync* inst)
{
  int32_T quotient;
  uint32_T absNumerator;
  uint32_T absDenominator;
  uint32_T tempAbsQuotient;
  uint32_T quotientNeedsNegation;
  if (denominator == 0) {
    quotient = numerator >= 0 ? MAX_int32_T : MIN_int32_T;

    /* Divide by zero handler */
  } else {
    absNumerator = (uint32_T)(numerator >= 0 ? numerator : -numerator);
    absDenominator = (uint32_T)(denominator >= 0 ? denominator : -denominator);
    quotientNeedsNegation = ((numerator < 0) != (denominator < 0));
    tempAbsQuotient = absNumerator / absDenominator;
    if (quotientNeedsNegation) {
      absNumerator %= absDenominator;
      if (absNumerator > 0) {
        tempAbsQuotient += (uint32_T)1;
      }
    }

    quotient = quotientNeedsNegation ? -(int32_T)tempAbsQuotient : (int32_T)
      tempAbsQuotient;
  }

  return quotient;
}

/* Model step function */
void FSync_step(struct BlockIO_FSync *FSync_B, struct D_Work_FSync *FSync_DWork,
                ExternalOutputs_FSync *FSync_Y, struct fFSync* inst)
{
  /* local block i/o variables */
  int16_T rtb_DataTypeConversion;
  int16_T rtb_DataTypeConversion1[2];
  int16_T rtb_DataTypeConversion2[2];
  uint8_T rtb_LookupTableDynamic;
  boolean_T rtb_LogicalOperator_o;
  uint8_T iNum_SkipMin;
  real32_T S;
  real32_T gk;
  boolean_T b;
  boolean_T c;
  boolean_T e;
  boolean_T f;
  boolean_T g;
  boolean_T h;
  boolean_T k;
  boolean_T l;
  real32_T rtb_Divide;
  int8_T rtb_Switch2;
  int8_T rtb_Abs;
  int8_T rtb_DataTypeConversion9;
  real32_T rtb_Switch1;
  boolean_T rtb_RelationalOperator_pw;
  real32_T rtb_Switch;
  real32_T rtb_Add1;
  boolean_T rtb_bEna;
  boolean_T rtb_bSetReached;
  uint32_T qY;
  int32_T tmp;

  /* S-Function (bur_bus_in): '<Root>/Bus Input' */
  FSync_B->BusInput = inst->In;

  /* S-Function (bur_bus_in): '<Root>/Bus Input1' */
  FSync_B->BusInput1 = inst->Perm;

  /* S-Function (bur_bus_in): '<Root>/Bus Input2' */
  FSync_B->BusInput2 = inst->Para;

  /* MATLAB Function: '<Root>/Skipfire_active' */
  /* MATLAB Function 'Skipfire_active': '<S7>:1' */
  /* % enable Sync function */
  if (FSync_B->BusInput.rN_Eng >= FSync_B->BusInput1.rN_enableNorm *
      FSync_B->BusInput2.rN_EngNom) {
    /* '<S7>:1:14' */
    /* '<S7>:1:15' */
    FSync_DWork->ssr = TRUE;
  }

  if (FSync_B->BusInput.rN_Eng >= FSync_B->BusInput1.rN_idleNorm *
      FSync_B->BusInput2.rN_EngNom) {
    /* '<S7>:1:18' */
    /* '<S7>:1:19' */
    FSync_DWork->ssr_Set = TRUE;
  }

  if (FSync_B->BusInput.bGCB_ON || (FSync_B->BusInput.rN_Eng < 100.0F)) {
    /* '<S7>:1:22' */
    /* '<S7>:1:23' */
    FSync_DWork->ssr = FALSE;

    /* '<S7>:1:24' */
    FSync_DWork->ssr_Set = FALSE;
  }

  /* '<S7>:1:28' */
  rtb_bEna = FSync_DWork->ssr;

  /* '<S7>:1:29' */
  rtb_bSetReached = FSync_DWork->ssr_Set;

  /* End of MATLAB Function: '<Root>/Skipfire_active' */

  /* DataTypeConversion: '<S5>/Data Type Conversion' incorporates:
   *  Gain: '<S5>/Gain'
   */
  S = (real32_T)fmod((real32_T)floor(10.0F * FSync_B->BusInput.rT_EO), 65536.0F);
  rtb_DataTypeConversion = (int16_T)(S < 0.0F ? (int16_T)-(int16_T)(uint16_T)-S :
                                     (int16_T)(uint16_T)S);

  /* DataTypeConversion: '<S5>/Data Type Conversion1' incorporates:
   *  BusSelector: '<S5>/Bus Selector1'
   *  Gain: '<S5>/Gain1'
   */
  S = (real32_T)fmod((real32_T)floor(10.0F * FSync_B->BusInput1.rT_Cold),
                     65536.0F);
  rtb_DataTypeConversion1[0] = (int16_T)(S < 0.0F ? (int16_T)-(int16_T)(uint16_T)
    -S : (int16_T)(uint16_T)S);
  S = (real32_T)fmod((real32_T)floor(10.0F * FSync_B->BusInput1.rT_Warm),
                     65536.0F);
  rtb_DataTypeConversion1[1] = (int16_T)(S < 0.0F ? (int16_T)-(int16_T)(uint16_T)
    -S : (int16_T)(uint16_T)S);

  /* DataTypeConversion: '<S5>/Data Type Conversion2' incorporates:
   *  BusSelector: '<S5>/Bus Selector1'
   */
  rtb_DataTypeConversion2[0] = FSync_B->BusInput1.iNum_SkipCyl_Cold;
  rtb_DataTypeConversion2[1] = FSync_B->BusInput1.iNum_SkipCyl_Warm;

  /* Dynamic Look-Up Table Block: '<S5>/Lookup Table Dynamic'
   * Input0  Data Type:  Integer        S16
   * Input1  Data Type:  Integer        S16
   * Input2  Data Type:  Integer        S16
   * Output0 Data Type:  Integer        U8
   * Lookup Method: Linear_Endpoint
   *
   */
  LookUp_U8S16_S16( &(rtb_LookupTableDynamic), rtb_DataTypeConversion2,
                   rtb_DataTypeConversion, rtb_DataTypeConversion1, 1U, inst);

  /* Switch: '<S9>/Switch1' incorporates:
   *  Constant: '<S13>/Constant'
   *  Logic: '<S9>/Logical Operator3'
   *  Product: '<S9>/Divide1'
   *  RelationalOperator: '<S13>/Compare'
   */
  if (FSync_B->BusInput1.bF_act_ena && (FSync_B->BusInput.iIdx_SyOMSS > 0)) {
    /* Switch: '<S15>/Switch' incorporates:
     *  Abs: '<S15>/Abs'
     *  RelationalOperator: '<S15>/Relational Operator'
     */
    if (1.0F >= (real32_T)fabs(FSync_B->BusInput2.rF_Nom)) {
      S = 1.0F;
    } else {
      S = FSync_B->BusInput2.rF_Nom;
    }

    /* End of Switch: '<S15>/Switch' */
    rtb_Switch1 = FSync_B->BusInput.rF_MMD * FSync_B->BusInput2.rN_EngNom / S;
  } else {
    rtb_Switch1 = FSync_B->BusInput.rN_Eng;
  }

  /* End of Switch: '<S9>/Switch1' */

  /* Switch: '<S16>/Switch' incorporates:
   *  Abs: '<S16>/Abs'
   *  BusSelector: '<S9>/Bus Selector'
   *  RelationalOperator: '<S16>/Relational Operator'
   */
  if (1.0F >= (real32_T)fabs(FSync_B->BusInput2.rF_Nom)) {
    S = 1.0F;
  } else {
    S = FSync_B->BusInput2.rF_Nom;
  }

  /* End of Switch: '<S16>/Switch' */

  /* Product: '<S9>/Divide' */
  rtb_Divide = FSync_B->BusInput.rF_MMD_BusBar / S *
    FSync_B->BusInput2.rN_EngNom;

  /* Outputs for Atomic SubSystem: '<S9>/Filter' */
  /* RelationalOperator: '<S17>/Relational Operator' incorporates:
   *  Constant: '<S17>/Constant'
   */
  rtb_RelationalOperator_pw = (FSync_B->BusInput1.rTi_FiltF > 0.0F);

  /* Logic: '<S17>/Logical Operator' incorporates:
   *  Logic: '<S17>/Logical Operator1'
   */
  rtb_LogicalOperator_o = (FSync_B->BusInput.bReset ||
    (!rtb_RelationalOperator_pw));

  /* DiscreteIntegrator: '<S17>/Discrete-Time Integrator' */
  if (FSync_DWork->DiscreteTimeIntegrator_IC_LOADI != 0) {
    FSync_DWork->DiscreteTimeIntegrator_DSTATE = FSync_B->BusInput2.rN_EngNom;
  }

  if (rtb_LogicalOperator_o || (FSync_DWork->DiscreteTimeIntegrator_PrevRese !=
       0)) {
    FSync_DWork->DiscreteTimeIntegrator_DSTATE = FSync_B->BusInput2.rN_EngNom;
  }

  /* Switch: '<S17>/Switch' incorporates:
   *  DiscreteIntegrator: '<S17>/Discrete-Time Integrator'
   */
  if (rtb_RelationalOperator_pw) {
    rtb_Switch = FSync_DWork->DiscreteTimeIntegrator_DSTATE;
  } else {
    rtb_Switch = rtb_Divide;
  }

  /* End of Switch: '<S17>/Switch' */

  /* Update for DiscreteIntegrator: '<S17>/Discrete-Time Integrator' */
  FSync_DWork->DiscreteTimeIntegrator_IC_LOADI = 0U;

  /* Switch: '<S21>/Switch' incorporates:
   *  Abs: '<S21>/Abs'
   *  RelationalOperator: '<S21>/Relational Operator'
   */
  if (2.22044605E-16F >= (real32_T)fabs(FSync_B->BusInput1.rTi_FiltF)) {
    S = 2.22044605E-16F;
  } else {
    S = FSync_B->BusInput1.rTi_FiltF;
  }

  /* End of Switch: '<S21>/Switch' */

  /* Update for DiscreteIntegrator: '<S17>/Discrete-Time Integrator' incorporates:
   *  DiscreteIntegrator: '<S17>/Discrete-Time Integrator'
   *  Product: '<S17>/Divide4'
   *  Sum: '<S17>/Sum4'
   */
  FSync_DWork->DiscreteTimeIntegrator_DSTATE += (rtb_Divide -
    FSync_DWork->DiscreteTimeIntegrator_DSTATE) / S * 0.01F;
  if (rtb_LogicalOperator_o) {
    FSync_DWork->DiscreteTimeIntegrator_PrevRese = 1;
  } else {
    FSync_DWork->DiscreteTimeIntegrator_PrevRese = 0;
  }

  /* End of Outputs for SubSystem: '<S9>/Filter' */

  /* Switch: '<S9>/Switch2' incorporates:
   *  Constant: '<S11>/Constant'
   *  Constant: '<S9>/Constant'
   *  Logic: '<S9>/Logical Operator1'
   *  RelationalOperator: '<S11>/Compare'
   */
  if ((FSync_B->BusInput.iIdx_SyOMSS > 0) && FSync_B->BusInput2.bFastSync) {
    rtb_Switch2 = FSync_B->BusInput1.iCtrSel;
  } else {
    rtb_Switch2 = 1;
  }

  /* End of Switch: '<S9>/Switch2' */

  /* Switch: '<S9>/Switch' incorporates:
   *  BusSelector: '<S9>/Bus Selector'
   *  Constant: '<S14>/Constant'
   *  Constant: '<S9>/Constant1'
   *  Logic: '<S9>/Logical Operator'
   *  Product: '<S9>/Product1'
   *  RelationalOperator: '<S14>/Compare'
   *  RelationalOperator: '<S9>/Relational Operator'
   */
  if (FSync_B->BusInput1.bSpeedSet_ena || (FSync_B->BusInput.iIdx_SyOMSS == 0) ||
      (FSync_B->BusInput.rF_MMD_BusBar < 0.5F * FSync_B->BusInput2.rF_Nom)) {
    rtb_Switch = FSync_B->BusInput2.rN_EngNom;
  }

  /* End of Switch: '<S9>/Switch' */

  /* Switch: '<S9>/Switch4' incorporates:
   *  Constant: '<S10>/Constant'
   *  Constant: '<S12>/Constant'
   *  Constant: '<S9>/Const_0'
   *  Logic: '<S9>/Logical Operator2'
   *  RelationalOperator: '<S10>/Compare'
   *  RelationalOperator: '<S12>/Compare'
   */
  if ((FSync_B->BusInput.iIdx_SyOMSS > 0) && (rtb_Switch2 == 1)) {
    S = FSync_B->BusInput2.rN_Offs_Sync;
  } else {
    S = 0.0F;
  }

  /* End of Switch: '<S9>/Switch4' */

  /* Sum: '<S9>/Add1' */
  rtb_Add1 = rtb_Switch + S;

  /* Abs: '<S9>/Abs' */
  if (FSync_B->BusInput1.iNum_SkipCylLim_P < 0) {
    rtb_Abs = (int8_T)-FSync_B->BusInput1.iNum_SkipCylLim_P;
  } else {
    rtb_Abs = FSync_B->BusInput1.iNum_SkipCylLim_P;
  }

  /* End of Abs: '<S9>/Abs' */

  /* Product: '<S9>/Product' incorporates:
   *  Sum: '<S9>/Add'
   */
  S = (rtb_Switch1 - rtb_Add1) * FSync_B->BusInput1.rGain_P;

  /* DataTypeConversion: '<S9>/Data Type Conversion9' */
  if (S < 0.0F) {
    S = (real32_T)ceil(S);
  } else {
    S = (real32_T)floor(S);
  }

  S = (real32_T)fmod(S, 256.0F);
  rtb_DataTypeConversion9 = (int8_T)(S < 0.0F ? (int8_T)-(int8_T)(uint8_T)-S :
    (int8_T)(uint8_T)S);

  /* End of DataTypeConversion: '<S9>/Data Type Conversion9' */

  /* Switch: '<S18>/Switch2' incorporates:
   *  RelationalOperator: '<S18>/LowerRelop1'
   */
  if (!(rtb_DataTypeConversion9 > rtb_Abs)) {
    /* Gain: '<S9>/Gain2' */
    rtb_Abs = (int8_T)-rtb_Abs;

    /* Switch: '<S18>/Switch' incorporates:
     *  RelationalOperator: '<S18>/UpperRelop'
     */
    if (!(rtb_DataTypeConversion9 < rtb_Abs)) {
      rtb_Abs = rtb_DataTypeConversion9;
    }

    /* End of Switch: '<S18>/Switch' */
  }

  /* End of Switch: '<S18>/Switch2' */

  /* MATLAB Function: '<Root>/SkipFireCtrl' incorporates:
   *  Gain: '<S9>/Conv rad'
   *  Product: '<S8>/Product1'
   *  SampleTimeMath: '<S8>/Weighted Sample Time'
   *
   * About '<S8>/Weighted Sample Time':
   *  y = K where K = 1 / ( w * Ts )
   */
  iNum_SkipMin = FSync_B->BusInput1.iNum_SkipMin;

  /* MATLAB Function 'SkipFireCtrl': '<S6>:1' */
  /* % init */
  if ((!FSync_DWork->cyl_skipped_not_empty) || (!rtb_bEna)) {
    /* '<S6>:1:14' */
    /* '<S6>:1:15' */
    FSync_DWork->cyl_skipped = 0U;
    FSync_DWork->cyl_skipped_not_empty = TRUE;

    /* '<S6>:1:16' */
    FSync_DWork->skipcounter = 0U;

    /* '<S6>:1:17' */
    FSync_DWork->bSkipDrehz_O = FALSE;

    /* '<S6>:1:18' */
    FSync_DWork->bSkipDrehz_U = FALSE;

    /* '<S6>:1:19' */
    FSync_DWork->Count_Switch = 0U;

    /* '<S6>:1:20' */
    FSync_DWork->No_Access = FALSE;

    /* '<S6>:1:21' */
    FSync_DWork->rN_Set_old = 0.0F;
  }

  /* % switch to ctrl 1 after a certain time */
  if (rtb_bSetReached) {
    /* '<S6>:1:26' */
    if (((real32_T)FSync_DWork->Count_Switch < FSync_B->BusInput1.rTi_FastSync *
         100.0F) && (rtb_Switch2 > 1)) {
      /* '<S6>:1:27' */
      /* '<S6>:1:28' */
      qY = (uint32_T)FSync_DWork->Count_Switch + 1U;
      if (qY > 65535U) {
        qY = 65535U;
      }

      FSync_DWork->Count_Switch = (uint16_T)qY;

      /* '<S6>:1:29' */
      FSync_B->bEnabled = TRUE;

      /* '<S6>:1:30' */
      FSync_DWork->No_Access = FALSE;
    } else if (!FSync_DWork->No_Access) {
      /* '<S6>:1:31' */
      /* '<S6>:1:32' */
      rtb_Switch2 = 1;

      /* '<S6>:1:33' */
      FSync_DWork->cyl_skipped = rtb_LookupTableDynamic;

      /* '<S6>:1:34' */
      FSync_DWork->No_Access = TRUE;

      /* '<S6>:1:35' */
      FSync_B->bEnabled = FSync_B->BusInput1.bStdCtrl;

      /*  switch to structured text standard controller if bStdCtrl is not set */
    } else {
      /* '<S6>:1:37' */
      rtb_Switch2 = 1;

      /* '<S6>:1:38' */
      FSync_B->bEnabled = FSync_B->BusInput1.bStdCtrl;
    }
  } else {
    /* '<S6>:1:41' */
    iNum_SkipMin = 0U;

    /* '<S6>:1:42' */
    FSync_B->bEnabled = TRUE;
  }

  if (FSync_DWork->skipcounter < 2000) {
    /* '<S6>:1:47' */
    /* '<S6>:1:48' */
    qY = (uint32_T)FSync_DWork->skipcounter + 1U;
    if (qY > 65535U) {
      qY = 65535U;
    }

    FSync_DWork->skipcounter = (uint16_T)qY;
  } else {
    /* '<S6>:1:50' */
    FSync_DWork->skipcounter = 0U;
  }

  /* % Modified law */
  /* '<S6>:1:56' */
  rtb_Divide = rtb_Switch1 - rtb_Add1;

  /* '<S6>:1:57' */
  rtb_Switch = 0.0174532924F * FSync_B->BusInput.rAng_MMD_Diff -
    FSync_B->BusInput1.rAngleSetDeg * 3.14159274F / 180.0F;

  /* '<S6>:1:59' */
  S = 0.5F * rtb_Divide * (real32_T)fabs(rtb_Divide) * 3.0F * 3.14159274F /
    30.0F * 3.0F * 3.14159274F / 30.0F + rtb_Switch;
  if ((0.5F * rtb_Divide * rtb_Divide * 3.0F * 3.14159274F / 30.0F * 3.0F *
       3.14159274F / 30.0F + rtb_Switch == 0.0F) && (rtb_Divide >= 0.0F)) {
    /* '<S6>:1:60' */
    b = TRUE;
  } else {
    /* '<S6>:1:60' */
    b = FALSE;
  }

  /*  x2: speed, x1: angle gamma minus */
  if ((-0.5F * rtb_Divide * rtb_Divide * 3.0F * 3.14159274F / 30.0F * 3.0F *
       3.14159274F / 30.0F + rtb_Switch == 0.0F) && (rtb_Divide <= 0.0F)) {
    /* '<S6>:1:61' */
    c = TRUE;
  } else {
    /* '<S6>:1:61' */
    c = FALSE;
  }

  /*  gamma plus */
  /*  why not using direct S1 ??? */
  /*  why not using direct S2 ??? */
  /* '<S6>:1:64' */
  /*  x2 */
  /*  x1                                                                              % not used, delete ??? */
  if ((S <= FSync_B->BusInput1.rRelaxAngleDeg * 3.14159274F / 180.0F) && (S >=
       -FSync_B->BusInput1.rRelaxAngleDeg * 3.14159274F / 180.0F) &&
      (-rtb_Divide < 0.0F)) {
    /* '<S6>:1:66' */
    rtb_RelationalOperator_pw = TRUE;
  } else {
    /* '<S6>:1:66' */
    rtb_RelationalOperator_pw = FALSE;
  }

  if ((S <= FSync_B->BusInput1.rRelaxAngleDeg * 3.14159274F / 180.0F) && (S >=
       -FSync_B->BusInput1.rRelaxAngleDeg * 3.14159274F / 180.0F) &&
      (-rtb_Divide > 0.0F)) {
    /* '<S6>:1:67' */
    e = TRUE;
  } else {
    /* '<S6>:1:67' */
    e = FALSE;
  }

  /* '<S6>:1:68' */
  /* '<S6>:1:69' */
  /* '<S6>:1:70' */
  if ((-0.5F * rtb_Divide * rtb_Divide * 3.0F * 3.14159274F / 30.0F * 3.0F *
       3.14159274F / 30.0F + rtb_Switch == FSync_B->BusInput1.rRelaxAngleDeg *
       3.14159274F / 180.0F) && (-rtb_Divide < 0.0F)) {
    /* '<S6>:1:71' */
    f = TRUE;
  } else {
    /* '<S6>:1:71' */
    f = FALSE;
  }

  if ((-FSync_B->BusInput1.rRelaxAngleDeg * 3.14159274F / 180.0F == S) &&
      (-rtb_Divide > 0.0F)) {
    /* '<S6>:1:72' */
    g = TRUE;
  } else {
    /* '<S6>:1:72' */
    g = FALSE;
  }

  if (rtb_RelationalOperator_pw || (S < -FSync_B->BusInput1.rRelaxAngleDeg *
       3.14159274F / 180.0F)) {
    /* '<S6>:1:66' */
    /* '<S6>:1:73' */
    h = TRUE;
  } else {
    /* '<S6>:1:73' */
    h = FALSE;
  }

  if (e || (S > FSync_B->BusInput1.rRelaxAngleDeg * 3.14159274F / 180.0F)) {
    /* '<S6>:1:67' */
    /* '<S6>:1:74' */
    rtb_RelationalOperator_pw = TRUE;
  } else {
    /* '<S6>:1:74' */
    rtb_RelationalOperator_pw = FALSE;
  }

  /*  k->inf, time optimal, k->0 fuel optimal */
  /* '<S6>:1:76' */
  gk = (FSync_B->BusInput1.rWeightFuel + 4.0F) / (2.0F *
    FSync_B->BusInput1.rWeightFuel);
  if ((S >= 0.0F) && (gk * rtb_Divide * (real32_T)fabs(rtb_Divide) * 3.0F *
                      3.14159274F / 30.0F * 3.0F * 3.14159274F / 30.0F +
                      rtb_Switch > 0.0F)) {
    /* '<S6>:1:77' */
    e = TRUE;
  } else {
    /* '<S6>:1:77' */
    e = FALSE;
  }

  /*  not used, delete ??? */
  if ((S <= 0.0F) && (gk * rtb_Divide * (real32_T)fabs(rtb_Divide) * 3.0F *
                      3.14159274F / 30.0F * 3.0F * 3.14159274F / 30.0F +
                      rtb_Switch < 0.0F)) {
    /* '<S6>:1:79' */
    k = TRUE;
  } else {
    /* '<S6>:1:79' */
    k = FALSE;
  }

  if ((S > 0.0F) && (gk * rtb_Divide * (real32_T)fabs(rtb_Divide) * 3.0F *
                     3.14159274F / 30.0F * 3.0F * 3.14159274F / 30.0F +
                     rtb_Switch <= 0.0F)) {
    /* '<S6>:1:80' */
    l = TRUE;
  } else {
    /* '<S6>:1:80' */
    l = FALSE;
  }

  /* '<S6>:1:81' */
  rtb_Divide = 10.0F * rtb_Divide * 3.0F * 3.14159274F / 30.0F * 3.0F *
    3.14159274F / 30.0F + rtb_Switch;

  /* % Change Selector */
  /* '<S6>:1:85' */
  switch (rtb_Switch2) {
   case 1:
    /*  Std skip firing */
    if ((rtb_Switch1 > rtb_Add1 + FSync_B->BusInput1.rN_SetTol) &&
        (FSync_DWork->cyl_skipped < 18) && rtb_bSetReached &&
        ((FSync_DWork->skipcounter > FSync_B->BusInput1.iSkipCounterLimit) ||
         FSync_DWork->bSkipDrehz_U)) {
      /* '<S6>:1:87' */
      /* Sid: prohibit entering if counter below limit, min dwell time in skip mode time optimal */
      /* '<S6>:1:88' */
      tmp = (int32_T)((uint32_T)FSync_DWork->cyl_skipped + 1U);
      if ((uint32_T)tmp > 255U) {
        tmp = 255;
      }

      FSync_DWork->cyl_skipped = (uint8_T)tmp;

      /*  increase mode */
      /* '<S6>:1:89' */
      FSync_DWork->skipcounter = 0U;

      /* '<S6>:1:90' */
      FSync_DWork->bSkipDrehz_O = TRUE;

      /* '<S6>:1:91' */
      FSync_DWork->bSkipDrehz_U = FALSE;
    } else {
      if ((rtb_Switch1 < rtb_Add1 - FSync_B->BusInput1.rN_SetTol) &&
          (FSync_DWork->cyl_skipped > 0) && rtb_bSetReached &&
          ((FSync_DWork->skipcounter > FSync_B->BusInput1.iSkipCounterLimit) ||
           FSync_DWork->bSkipDrehz_O)) {
        /* '<S6>:1:92' */
        /*  Cyl 1 and 11 are prmanently fired --> max 18 Cylinders skipped */
        /* '<S6>:1:93' */
        qY = (uint32_T)FSync_DWork->cyl_skipped - 1U;
        if (qY > FSync_DWork->cyl_skipped) {
          qY = 0U;
        }

        FSync_DWork->cyl_skipped = (uint8_T)(int32_T)qY;

        /*  decrease mode */
        /* '<S6>:1:94' */
        FSync_DWork->skipcounter = 0U;

        /* '<S6>:1:95' */
        FSync_DWork->bSkipDrehz_O = FALSE;

        /* '<S6>:1:96' */
        FSync_DWork->bSkipDrehz_U = TRUE;
      }
    }
    break;

   case 2:
    /*  Time optimal */
    if ((S > FSync_B->BusInput1.rHystOptimal) || (b && rtb_bEna)) {
      /* '<S6>:1:100' */
      /* '<S6>:1:60' */
      /* '<S6>:1:100' */
      /* '<S6>:1:101' */
      FSync_DWork->cyl_skipped = FSync_B->BusInput1.iNum_SkipMax;

      /*  increase mode */
      /* '<S6>:1:102' */
      FSync_DWork->skipcounter = 0U;

      /* '<S6>:1:103' */
      FSync_DWork->bSkipDrehz_O = TRUE;

      /* '<S6>:1:104' */
      FSync_DWork->bSkipDrehz_U = FALSE;
    } else {
      if ((S < -FSync_B->BusInput1.rHystOptimal) || (c && rtb_bEna)) {
        /* '<S6>:1:105' */
        /* '<S6>:1:61' */
        /* '<S6>:1:105' */
        /* '<S6>:1:106' */
        FSync_DWork->cyl_skipped = iNum_SkipMin;

        /*  decrease mode */
        /* '<S6>:1:107' */
        FSync_DWork->skipcounter = 0U;

        /* '<S6>:1:108' */
        FSync_DWork->bSkipDrehz_O = FALSE;

        /* '<S6>:1:109' */
        FSync_DWork->bSkipDrehz_U = TRUE;
      }
    }
    break;

   case 3:
    /*  Time optimal with constraints on the angle */
    if ((rtb_RelationalOperator_pw || g) && rtb_bEna) {
      /* '<S6>:1:74' */
      /* '<S6>:1:72' */
      /* '<S6>:1:113' */
      /* '<S6>:1:114' */
      FSync_DWork->cyl_skipped = FSync_B->BusInput1.iNum_SkipMax;

      /*  increase mode */
      /* '<S6>:1:115' */
      FSync_DWork->skipcounter = 0U;

      /* '<S6>:1:116' */
      FSync_DWork->bSkipDrehz_O = TRUE;

      /* '<S6>:1:117' */
      FSync_DWork->bSkipDrehz_U = FALSE;
    } else {
      if ((h || f) && rtb_bEna) {
        /* '<S6>:1:73' */
        /* '<S6>:1:71' */
        /* '<S6>:1:118' */
        /* '<S6>:1:119' */
        FSync_DWork->cyl_skipped = iNum_SkipMin;

        /*  decrease mode */
        /* '<S6>:1:120' */
        FSync_DWork->skipcounter = 0U;

        /* '<S6>:1:121' */
        FSync_DWork->bSkipDrehz_O = FALSE;

        /* '<S6>:1:122' */
        FSync_DWork->bSkipDrehz_U = TRUE;
      }
    }
    break;

   case 4:
    /*  Fuel and time optimal */
    if (e && rtb_bEna) {
      /* '<S6>:1:77' */
      /* '<S6>:1:126' */
      /* '<S6>:1:127' */
      FSync_DWork->cyl_skipped = FSync_B->BusInput1.iNum_SkipMax;

      /*  increase mode */
      /* '<S6>:1:128' */
      FSync_DWork->skipcounter = 0U;

      /* '<S6>:1:129' */
      FSync_DWork->bSkipDrehz_O = TRUE;

      /* '<S6>:1:130' */
      FSync_DWork->bSkipDrehz_U = FALSE;
    } else {
      if (k && rtb_bEna) {
        /* '<S6>:1:79' */
        /* '<S6>:1:131' */
        /*  use with averaging controller */
        /* '<S6>:1:132' */
        FSync_DWork->cyl_skipped = iNum_SkipMin;

        /*  decrease mode */
        /* '<S6>:1:133' */
        FSync_DWork->skipcounter = 0U;

        /* '<S6>:1:134' */
        FSync_DWork->bSkipDrehz_O = FALSE;

        /* '<S6>:1:135' */
        FSync_DWork->bSkipDrehz_U = TRUE;

        /*  elseif(H2)        % delete ??? */
        /*      cyl_skipped=cyl_skipped+1; */
        /*  elseif(H4) */
        /*      cyl_skipped=cyl_skipped-1; */
      }
    }
    break;

   case 5:
    /*  Modified skip firing */
    if ((rtb_Divide > 0.0F) && (FSync_DWork->cyl_skipped < 18) && rtb_bEna &&
        ((FSync_DWork->skipcounter > FSync_B->BusInput1.iSkipCounterLimit) ||
         FSync_DWork->bSkipDrehz_U)) {
      /* '<S6>:1:143' */
      /* Sid: prohibit entering if counter below limit, min dwell time in skip mode time optimal */
      /* '<S6>:1:144' */
      tmp = (int32_T)((uint32_T)FSync_DWork->cyl_skipped + 1U);
      if ((uint32_T)tmp > 255U) {
        tmp = 255;
      }

      FSync_DWork->cyl_skipped = (uint8_T)tmp;

      /*  increase mode */
      /* '<S6>:1:145' */
      FSync_DWork->skipcounter = 0U;

      /* '<S6>:1:146' */
      FSync_DWork->bSkipDrehz_O = TRUE;

      /* '<S6>:1:147' */
      FSync_DWork->bSkipDrehz_U = FALSE;
    } else {
      if ((rtb_Divide < 0.0F) && (FSync_DWork->cyl_skipped > 0) && rtb_bEna &&
          ((FSync_DWork->skipcounter > FSync_B->BusInput1.iSkipCounterLimit) ||
           FSync_DWork->bSkipDrehz_O)) {
        /* '<S6>:1:148' */
        /*  Cyl 1 and 11 are prmanently fired --> max 18 Cylinders skipped */
        /* '<S6>:1:149' */
        qY = (uint32_T)FSync_DWork->cyl_skipped - 1U;
        if (qY > FSync_DWork->cyl_skipped) {
          qY = 0U;
        }

        FSync_DWork->cyl_skipped = (uint8_T)(int32_T)qY;

        /*  decrease mode */
        /* '<S6>:1:150' */
        FSync_DWork->skipcounter = 0U;

        /* '<S6>:1:151' */
        FSync_DWork->bSkipDrehz_O = FALSE;

        /* '<S6>:1:152' */
        FSync_DWork->bSkipDrehz_U = TRUE;
      }
    }
    break;

   default:
    if ((rtb_Switch1 > rtb_Add1 + FSync_B->BusInput1.rN_SetTol) &&
        (FSync_DWork->cyl_skipped < 18) && rtb_bEna &&
        ((FSync_DWork->skipcounter > FSync_B->BusInput1.iSkipCounterLimit) ||
         FSync_DWork->bSkipDrehz_U)) {
      /* '<S6>:1:156' */
      /* Sid: prohibit entering if counter below limit, min dwell time in skip mode time optimal */
      /* '<S6>:1:157' */
      tmp = (int32_T)((uint32_T)FSync_DWork->cyl_skipped + 1U);
      if ((uint32_T)tmp > 255U) {
        tmp = 255;
      }

      FSync_DWork->cyl_skipped = (uint8_T)tmp;

      /*  increase mode */
      /* '<S6>:1:158' */
      FSync_DWork->skipcounter = 0U;

      /* '<S6>:1:159' */
      FSync_DWork->bSkipDrehz_O = TRUE;

      /* '<S6>:1:160' */
      FSync_DWork->bSkipDrehz_U = FALSE;
    } else {
      if ((rtb_Switch1 < rtb_Add1 - FSync_B->BusInput1.rN_SetTol) &&
          (FSync_DWork->cyl_skipped > 0) && rtb_bEna &&
          ((FSync_DWork->skipcounter > FSync_B->BusInput1.iSkipCounterLimit) ||
           FSync_DWork->bSkipDrehz_O)) {
        /* '<S6>:1:161' */
        /*  Cyl 1 and 11 are prmanently fired --> max 18 Cylinders skipped */
        /* '<S6>:1:162' */
        qY = (uint32_T)FSync_DWork->cyl_skipped - 1U;
        if (qY > FSync_DWork->cyl_skipped) {
          qY = 0U;
        }

        FSync_DWork->cyl_skipped = (uint8_T)(int32_T)qY;

        /*  decrease mode */
        /* '<S6>:1:163' */
        FSync_DWork->skipcounter = 0U;

        /* '<S6>:1:164' */
        FSync_DWork->bSkipDrehz_O = FALSE;

        /* '<S6>:1:165' */
        FSync_DWork->bSkipDrehz_U = TRUE;
      }
    }
    break;
  }

  /* % Output */
  /*  fire all cylinders in case of setpoint increase */
  if (rtb_Add1 - FSync_DWork->rN_Set_old > 100.0F) {
    /* '<S6>:1:172' */
    /* '<S6>:1:173' */
    FSync_DWork->cyl_skipped = 0U;
  }

  /* '<S6>:1:175' */
  FSync_DWork->rN_Set_old = rtb_Add1;
  if (!rtb_bEna) {
    /* Outport: '<Root>/SkipCyl' */
    /* '<S6>:1:178' */
    /* '<S6>:1:179' */
    FSync_Y->SkipCyl = 0U;
  } else if (rtb_Switch2 == 1) {
    /* '<S6>:1:181' */
    /* '<S6>:1:182' */
    iNum_SkipMin = FSync_DWork->cyl_skipped;
    if (FSync_DWork->cyl_skipped > 127) {
      iNum_SkipMin = 127U;
    }

    tmp = iNum_SkipMin + rtb_Abs;
    if (tmp > 127) {
      tmp = 127;
    }

    rtb_DataTypeConversion9 = (int8_T)tmp;
    if ((int8_T)tmp < 0) {
      rtb_DataTypeConversion9 = 0;
    }

    /* Outport: '<Root>/SkipCyl' */
    FSync_Y->SkipCyl = (uint8_T)rtb_DataTypeConversion9;
  } else {
    /* Outport: '<Root>/SkipCyl' */
    /* '<S6>:1:184' */
    FSync_Y->SkipCyl = FSync_DWork->cyl_skipped;
  }

  /* % debugging */
  /* '<S6>:1:189' */
  FSync_Y->dbg.iSkipCounter = FSync_DWork->skipcounter;

  /* '<S6>:1:190' */
  FSync_Y->dbg.rSwitchSurf = S;

  /* '<S6>:1:191' */
  FSync_Y->dbg.Sf1 = c;

  /* '<S6>:1:192' */
  FSync_Y->dbg.Sf2 = b;

  /* '<S6>:1:193' */
  FSync_Y->dbg.H3 = k;

  /* '<S6>:1:194' */
  FSync_Y->dbg.H4 = l;

  /* '<S6>:1:195' */
  FSync_Y->dbg.rSmodSlid = rtb_Divide;

  /* '<S6>:1:196' */
  FSync_Y->dbg.iCounterSwitch = FSync_DWork->Count_Switch;

  /* '<S6>:1:197' */
  FSync_Y->dbg.bEna = rtb_bEna;

  /* '<S6>:1:198' */
  FSync_Y->dbg.iNskip_init = rtb_LookupTableDynamic;

  /* '<S6>:1:199' */
  FSync_Y->dbg.iCtrSel = rtb_Switch2;

  /* '<S6>:1:200' */
  FSync_Y->dbg.iNumSkipCyl_P = rtb_Abs;

  /* '<S6>:1:201' */
  FSync_Y->dbg.rN_Set = rtb_Add1;

  /* '<S6>:1:202' */
  FSync_Y->dbg.rN_Eng = rtb_Switch1;

  /* End of MATLAB Function: '<Root>/SkipFireCtrl' */

  /* S-Function (bur_bus_out): '<Root>/Bus Output1' */
  inst->dbg = FSync_Y->dbg;

  /* S-Function (bur_out): '<Root>/Output' */
  inst->iSkipCyl = FSync_Y->SkipCyl;

  /* S-Function (bur_out): '<Root>/Output3' */
  inst->bEnabled = FSync_B->bEnabled;

  /* UnitDelay: '<S4>/Unit Delay' */
  FSync_B->UnitDelay = FSync_DWork->UnitDelay_DSTATE;

  /* S-Function (bur_out): '<Root>/Output2' */
  inst->Version = FSync_B->UnitDelay;

  /* Update for UnitDelay: '<S4>/Unit Delay' */
  FSync_DWork->UnitDelay_DSTATE = 7U;
}

/* Model initialize function */
void FSync_initialize(struct D_Work_FSync *FSync_DWork, struct fFSync* inst)
{
  /* InitializeConditions for Atomic SubSystem: '<S9>/Filter' */
  /* InitializeConditions for DiscreteIntegrator: '<S17>/Discrete-Time Integrator' */
  FSync_DWork->DiscreteTimeIntegrator_IC_LOADI = 1U;

  /* End of InitializeConditions for SubSystem: '<S9>/Filter' */
}

/* Model terminate function */
void FSync_terminate(struct fFSync* inst)
{
  /* (no terminate code required) */
}

/*======================== TOOL VERSION INFORMATION ==========================*
 * MATLAB 8.0 (R2012b)20-Jul-2012                                             *
 * Simulink 8.0 (R2012b)20-Jul-2012                                           *
 * Simulink Coder 8.3 (R2012b)20-Jul-2012                                     *
 * Embedded Coder 6.3 (R2012b)20-Jul-2012                                     *
 * Stateflow 8.0 (R2012b)20-Jul-2012                                          *
 *============================================================================*/

/*======================= LICENSE IN USE INFORMATION =========================*
 * matlab                                                                     *
 * matlab_coder                                                               *
 * real-time_workshop                                                         *
 * rtw_embedded_coder                                                         *
 * simulink                                                                   *
 *============================================================================*/
```

#### fFSync.c
```c
/********************************************************************
 * COPYRIGHT -- Bernecker + Rainer Industrie-Elektronik Ges.m.b.H.
 ********************************************************************
 * Program: FSync
 * File: fFSync.c
 * Author: 105051359
 * Created: Mon Mar 13 15:42:43 2017
 ********************************************************************
 * Implementation of program FSync
 ********************************************************************
 * Generated with B&R Automation Studio Target for Simulink V4.2
 * (ERT based)
 ********************************************************************/
#include <bur/plctypes.h>
#include "FSync.h"
#include "rtwtypes.h"

/* Defines */
#define SS_TERMINATE 4
#define SS_OUTPUT 3
#define SS_INITIALIZE 2

/*  Data Types */

/**************************** GLOBAL DATA *************************************/
/*  Definitions */

/*  Declarations  */

/***************************** FILE SCOPE DATA ********************************/

/*************************** FUNCTIONS ****************************************/
#ifdef __cplusplus

unsigned long bur_heap_size = 6553500;

#endif

void fFSync(struct fFSync* inst)
{
  BlockIO_FSync *FSync_B = &(inst)->bur_BlockIO_FSync;
	D_Work_FSync *FSync_DWork = &(inst)->bur_D_Work_FSync;
	ExternalOutputs_FSync *FSync_Y = &(inst)->bur_ExternalOutputs_FSync;

  switch (inst->ssMethodType)
  {
   case SS_INITIALIZE:
    /* call model initialize function */
    FSync_initialize(FSync_DWork, inst);
    break;

   case SS_OUTPUT:
    /* call model step function */
    FSync_step(FSync_B, FSync_DWork, FSync_Y, inst);

    break;

   case SS_TERMINATE:
    /* call model terminate function */
    FSync_terminate(inst);
    break;
  }
}

/*****************************************************************************
   Function block sample time: 0.01s
 *****************************************************************************/

/*****************************************************************************
   B&R Automation Studio Target for Simulink Version: A4.5.1 (27-Jul-2015)
 *****************************************************************************/

/*======================== TOOL VERSION INFORMATION ==========================*
 * MATLAB 8.0 (R2012b)20-Jul-2012                                             *
 * Simulink 8.0 (R2012b)20-Jul-2012                                           *
 * Simulink Coder 8.3 (R2012b)20-Jul-2012                                     *
 * Embedded Coder 6.3 (R2012b)20-Jul-2012                                     *
 * Stateflow 8.0 (R2012b)20-Jul-2012                                          *
 *============================================================================*/

/*======================= LICENSE IN USE INFORMATION =========================*
 * matlab                                                                     *
 * matlab_coder                                                               *
 * real-time_workshop                                                         *
 * rtw_embedded_coder                                                         *
 * simulink                                                                   *
 *============================================================================*/
```

#### lib_properties.txt
```
For manual assignment to hardware configuration please
add the following additional include directories:

\Logical\MATLAB_includes\R2012b\

And the following additional build options:

-lm -D MODEL=FSync -D NUMST=1 -D NCSTATES=0 -D HAVESTDIO -D ONESTEPFCN=1 -D TERMFCN=1 -D MAT_FILE=0 -D MULTI_INSTANCE_CODE=1 -D INTEGER_CODE=0 -D MT=0 -D CLASSIC_INTERFACE=0 -D TID01EQ=0
```

### Library Logical/EngineController/Lib_EC/lLamStart (ANSIC)

#### lLamStart.fun
```iecst
FUNCTION_BLOCK fLamStart
  VAR_INPUT
    ssMethodType: SINT;
  END_VAR  VAR_INPUT
        Perm : tLamStart_PERM; (**)
  END_VAR
  VAR_INPUT
        Para : tLamStart_PARA; (**)
  END_VAR
  VAR_INPUT
        IN : tLamStart_IN; (**)
  END_VAR
 VAR_OUTPUT
        dbg : tLamStart_DBG; (**)
  END_VAR
  VAR_OUTPUT
        rLambda_start_idle : REAL; (**)
  END_VAR
  VAR_OUTPUT
        Version : UDINT; (**)
  END_VAR
	VAR
		bur_BlockIO_LamStart : BlockIO_LamStart;
	END_VAR
	VAR
		bur_D_Work_LamStart : D_Work_LamStart;
	END_VAR
	VAR
		bur_PrevZCSigStates_LamStart : PrevZCSigStates_LamStart;
	END_VAR
	VAR
		bur_ExternalOutputs_LamStart : ExternalOutputs_LamStart;
	END_VAR
END_FUNCTION_BLOCK
```

#### lLamStart.typ
```iecst
TYPE

   tLamStart_DBG : STRUCT
        rLambda_start : REAL; (**)
        rLambda_idle : REAL; (**)
        rLambda_start_raw : REAL; (**)
        rLamLim : REAL; (**)
    END_STRUCT;

   tLamStart_IN : STRUCT
        rN_Eng : REAL; (*Engine speed [rpm]*)
        rT_EO : REAL; (**)
        bGCB_ON : BOOL; (*Generator curcuit breaker ON [-]*)
        bReset : BOOL; (*Reset Filters [-]*)
    END_STRUCT;

   tLamStart_PARA : STRUCT
        rN_EngNom : REAL; (*Nominal engine speed [rpm]*)
        rLam_Start_Offs : REAL; (**)
    END_STRUCT;

   tLamStart_PERM : STRUCT
        rLamSlewRate : REAL; (*slew rate to ramp back to zero offset [1/s]*)
        rTi_idle : REAL; (*ramp back to zero offset after X sec in idle mode [s]*)
        rLamLoLim_N_x : ARRAY[0..2] OF REAL; (*Lower lambda limit lookup depending on engine speed [rpm]*)
        rLamLoLim_N_y : ARRAY[0..2] OF REAL; (*Lower lambda limit lookup depending on engine speed [-]*)
        rLowerOilTemp : REAL; (**)
        rHigherOilTemp : REAL; (**)
        rLowerOilLambda : REAL; (**)
        rHigherOilLambda : REAL; (**)
        refPoint_Lam_N_Offs_x : ARRAY[0..2] OF REAL; (**)
        refPoint_Lam_N_Offs_y : ARRAY[0..2] OF REAL; (**)
    END_STRUCT;
END_TYPE
TYPE
BlockIO_LamStart : STRUCT
	BusInput2 : tLamStart_PERM;
	BusInput : tLamStart_IN;
	BusConversion_InsertedFor_BusOu : tLamStart_DBG;
	BusInput1 : tLamStart_PARA;
	UnitDelay : UDINT;
END_STRUCT;
D_Work_LamStart : STRUCT
	Delay_DSTATE : REAL;
	DiscreteTimeIntegrator_DSTATE : REAL;
	UnitDelay_DSTATE : UDINT;
	UnitDelay2_DSTATE : BOOL;
	DiscreteTimeIntegrator_PrevRese : SINT;
	icLoad : USINT;
END_STRUCT;
PrevZCSigStates_LamStart : STRUCT
	Delay_Reset_ZCE : USINT;
END_STRUCT;
ExternalInputs_LamStart : STRUCT
	IN : tLamStart_IN;
	PARA : tLamStart_PARA;
	PERM : tLamStart_PERM;
END_STRUCT;
ExternalOutputs_LamStart : STRUCT
	rLambda_start_idle : REAL;
	dbg : tLamStart_DBG;
END_STRUCT;
END_TYPE
```

#### LamStart.h
```c
/********************************************************************
 * COPYRIGHT -- Bernecker + Rainer Industrie-Elektronik Ges.m.b.H.
 ********************************************************************
 * Program: LamStart
 * File: LamStart.h
 * Author: 105055527
 * Created: Thu May 18 17:26:11 2017
 ********************************************************************
 * Header for program LamStart
 ********************************************************************
 * Generated with B&R Automation Studio Target for Simulink V4.2
 * (ERT based)
 ********************************************************************/

#ifndef RTW_HEADER_LamStart_h_
#define RTW_HEADER_LamStart_h_
#ifndef LamStart_COMMON_INCLUDES_
# define LamStart_COMMON_INCLUDES_
#include <math.h>
#include "rtwtypes.h"
#endif                                 /* LamStart_COMMON_INCLUDES_ */

#include "LamStart_types.h"
#include "lLamStart.h"

/* Macros for accessing real-time model data structure */
#ifndef rtmGetErrorStatus
# define rtmGetErrorStatus(rtm)        ((void*) 0)
#endif

#ifndef rtmSetErrorStatus
# define rtmSetErrorStatus(rtm, val)   ((void) 0)
#endif

#ifndef rtmGetStopRequested
# define rtmGetStopRequested(rtm)      ((void*) 0)
#endif

#ifndef MIN
#define MIN(a,b)                       ((a) < (b) ? (a) : (b))
#endif

#ifndef MAX
#define MAX(a,b)                       ((a) > (b) ? (a) : (b))
#endif

/* Block signals (auto storage) */

/* Block states (auto storage) for system '<Root>' */

/* Zero-crossing (trigger) state */

/* External inputs (root inport signals with auto storage) */

/* External outputs (root outports fed by signals with auto storage) */

/* Model entry point functions */
extern void LamStart_initialize(D_Work_LamStart *LamStart_DWork,
  PrevZCSigStates_LamStart *LamStart_PrevZCSigState, struct fLamStart* inst);
extern void LamStart_step(BlockIO_LamStart *LamStart_B, D_Work_LamStart
  *LamStart_DWork, PrevZCSigStates_LamStart *LamStart_PrevZCSigState,
  ExternalOutputs_LamStart *LamStart_Y, struct fLamStart* inst);
extern void LamStart_terminate(struct fLamStart* inst);

/*-
 * The generated code includes comments that allow you to trace directly
 * back to the appropriate location in the model.  The basic format
 * is <system>/block_name, where system is the system number (uniquely
 * assigned by Simulink) and block_name is the name of the block.
 *
 * Use the MATLAB hilite_system command to trace the generated code back
 * to the model.  For example,
 *
 * hilite_system('<S3>')    - opens system 3
 * hilite_system('<S3>/Kp') - opens and selects block Kp which resides in S3
 *
 * Here is the system hierarchy for this model
 *
 * '<Root>' : 'LamStart'
 * '<S1>'   : 'LamStart/EC1'
 * '<S2>'   : 'LamStart/EC2'
 * '<S3>'   : 'LamStart/EC3'
 * '<S4>'   : 'LamStart/Info'
 * '<S5>'   : 'LamStart/Saturation Dynamic'
 * '<S6>'   : 'LamStart/enableStartLambda'
 * '<S7>'   : 'LamStart/enableStartLambda/Hysteresis'
 * '<S8>'   : 'LamStart/enableStartLambda/TON'
 * '<S9>'   : 'LamStart/enableStartLambda/rateLimit'
 * '<S10>'  : 'LamStart/enableStartLambda/TON/Data Type Conversion Inherited'
 * '<S11>'  : 'LamStart/enableStartLambda/rateLimit/Saturation Dynamic'
 */
#endif                                 /* RTW_HEADER_LamStart_h_ */
```

#### LamStart_private.h
```c
/********************************************************************
 * COPYRIGHT -- Bernecker + Rainer Industrie-Elektronik Ges.m.b.H.
 ********************************************************************
 * Program: LamStart
 * File: LamStart_private.h
 * Author: 105055527
 * Created: Thu May 18 17:26:11 2017
 ********************************************************************
 * Header for program LamStart
 ********************************************************************
 * Generated with B&R Automation Studio Target for Simulink V4.2
 * (ERT based)
 ********************************************************************/

#ifndef RTW_HEADER_LamStart_private_h_
#define RTW_HEADER_LamStart_private_h_
#include "rtwtypes.h"
#include <bur/plctypes.h>
#ifndef __RTWTYPES_H__
#error This file requires rtwtypes.h to be included
#else
#ifdef TMWTYPES_PREVIOUSLY_INCLUDED
#error This file requires rtwtypes.h to be included before tmwtypes.h
#else

/* Check for inclusion of an incorrect version of rtwtypes.h */
#ifndef RTWTYPES_ID_C08S16I32L32N32F1
#error This code was generated with a different "rtwtypes.h" than the file included
#endif                                 /* RTWTYPES_ID_C08S16I32L32N32F1 */
#endif                                 /* TMWTYPES_PREVIOUSLY_INCLUDED */
#endif                                 /* __RTWTYPES_H__ */

#ifndef MIN
#define MIN(a,b)                       ((a) < (b) ? (a) : (b))
#endif

#ifndef MAX
#define MAX(a,b)                       ((a) > (b) ? (a) : (b))
#endif

void BINARYSEARCH_real32_T(uint32_T *piLeft, uint32_T *piRght, real32_T u, const
  real32_T *pData, uint32_T iHi, struct fLamStart* inst);
void LookUp_real32_T_real32_T(real32_T *pY, const real32_T *pYData, real32_T u,
  const real32_T *pUData, uint32_T iHi, struct fLamStart* inst);

#endif                                 /* RTW_HEADER_LamStart_private_h_ */
```

#### LamStart_types.h
```c
/********************************************************************
 * COPYRIGHT -- Bernecker + Rainer Industrie-Elektronik Ges.m.b.H.
 ********************************************************************
 * Program: LamStart
 * File: LamStart_types.h
 * Author: 105055527
 * Created: Thu May 18 17:26:11 2017
 ********************************************************************
 * Header for program LamStart
 ********************************************************************
 * Generated with B&R Automation Studio Target for Simulink V4.2
 * (ERT based)
 ********************************************************************/

#ifndef RTW_HEADER_LamStart_types_h_
#define RTW_HEADER_LamStart_types_h_
#include "rtwtypes.h"
#ifndef MIN
#define MIN(a,b)                       ((a) < (b) ? (a) : (b))
#endif

#ifndef MAX
#define MAX(a,b)                       ((a) > (b) ? (a) : (b))
#endif

#endif                                 /* RTW_HEADER_LamStart_types_h_ */
```
